	//******************** SCHEDA IN AP200.8
	I_AP200_8 			AT %I*: ARRAY[1..16] OF BOOL;
	//I_FREE 				: bool; // 1 = FREE
	//I_FREE 				: bool; // 2 = FREE
	//I_FREE 				: bool; // 3 = FREE
	//I_FREE 				: bool; // 4 = FREE
	I_24VOK_PS308			: BOOL;	// 5 = Presenza 24V PS308
	I_24VOK_PS309			: BOOL;	// 6 = Presenza 24V PS309
	I_24VOK_JB314			: BOOL;	// 7 = Presenza 24V JB314
	I_24VOK_JB315			: BOOL;	// 8 = Presenza 24V JB315
	//I_PresenzaSupporto[5] : BOOL;	// 9 = 
	//I_PresenzaTelaio[5]	: BOOL;	// 10 = 
	//I_PresenzaCentrale[5]	: BOOL;	// 11 = 
	//I_PresenzaBundle[5] 	: BOOL; // 12 = 
	//I_PresenzaSupporto[6] : BOOL;	// 13 = 
	//I_PresenzaTelaio[6]	: BOOL;	// 14 = 
	//I_PresenzaCentrale[6]	: BOOL;	// 15 = 
	//I_PresenzaBundle[6] 	: BOOL; // 16 =

	//******************** SCHEDA IN SAFETY AP200.9		
	I_AP200_9	AT %I*: ARRAY[1..4] OF BOOL;
	I_RicevitoreConsensoVeicolo AT %I*: ARRAY[1..8] OF BOOL;
	//I_RicevitoreConsensoVeicolo[1]	: BOOL; // 1=
	//I_RicevitoreConsensoVeicolo[2] 	: BOOL; // 2=	
	//I_RicevitoreConsensoVeicolo[3]	: BOOL; // 3=	
	//I_RicevitoreConsensoVeicolo[4]	: BOOL; // 4=	
	
	//******************** SCHEDA IN SAFETY AP200.10		
	I_AP200_10	AT %I*: ARRAY[1..4] OF BOOL;
	I_RichiestaIngressoPS308 			AT %I* : BOOL; // 2 = Richiesta ingresso Pal PS308
	I_ResetRichiestaIngressoPS308 		AT %I* : BOOL; // 6 = Richiesta ingresso Pal PS308
	//I_BarrieraCentroDx_CH1			: BOOL; // 3=	
	//I_BarrieraCentroDx_CH2			: BOOL; // 4=	

	//******************** SCHEDA IN SAFETY AP201.2		
	I_AP201_2	AT %I*: ARRAY[1..4] OF BOOL;
	//I_FeedBackMarcia				: BOOL; // 1=
	I_ResetRichiestaIngressoPS309 				AT %I* : BOOL; // 6 = Richiesta ingresso Pal PS309
	//I_BarrieraInterna_CH1			: BOOL; // 3=	
	//I_BarrieraInterna_CH2			: BOOL; // 4=	

	//******************** SCHEDA OUT AP201.4
	O_AP201_4 			AT %Q*: ARRAY[1..16] OF BOOL;		
	O_SirenaAllarmiPal							: BOOL;	// 1 = Sirena Allarmi
	O_LampadaAutomaticoPal						: BOOL;	// 2 = Lampada AUtomatico
	O_LampadaAllarmiPal							: BOOL;	// 3 = Lampada Allarmi
	O_LampadaRichiestaIngressoPal				: BOOL;	// 4 = Lampada Richiesta Ingresso PAL 1
	O_ConsensoVeicolo 							: ARRAY[1..8] OF BOOL;
	//O_ConsensoVeicolo[1]						: BOOL;	// 5 =
	//O_ConsensoVeicolo[2]						: BOOL;	// 6 =
	//O_ConsensoVeicolo[3]						: BOOL;	// 7 =
	//O_ConsensoVeicolo[4]						: BOOL;	// 8 =
	O_LampadaPulsanteCicloPalConsolle 			: BOOL;	//9 = Lampada Pulsante Ciclo Pallettizzatore
	O_LampadaPulsanteRichiestaIngressoConsolle 	: BOOL; //10 = Lampada Pulsante richiesta ingresso PS305
	O_LampadaPulsanteMarciaPalConsolle 			: BOOL;	//11 = Lampada Pulsante Marcia Pal 1 Consolle
	O_LampadaPulsanteRichiestaIngressoPS306 	: BOOL; //12 = Lampada Pulsante richiesta ingresso PS306
	O_LampadaPulsanteRichiestaIngressoPS307		: BOOL; //13 = Lampada Pulsante richiesta ingresso PS307
	O_LampadaPulsanteRichiestaIngressoPS308 	: BOOL; //14 = Lampada Pulsante richiesta ingresso PS308
	O_LampadaPulsanteRichiestaIngressoPS309		: BOOL; //15 = Lampada Pulsante richiesta ingresso PS309
	//FREE 										: BOOL; //16 =

	//******************** SCHEDA OUT SAFETY AP201.5		
	O_AP201_5	AT %Q*: ARRAY[1..4] OF BOOL;  			I_AP201_5 AT %I*: ARRAY[1..4] OF BOOL;//Appoggio
	//O_MarciaPal	: BOOL; // CH1=
	//FREE			: BOOL; // CH2=	
	//FREE			: BOOL; // CH3=	
	//FREE			: BOOL; // CH4=	
	
	//******************** SCHEDA OUT AP201.6	
	O_AP201_6 						AT %Q*: ARRAY[1..16] OF BOOL;
	
	O_LampadaIngressoVietatoPS306 	: BOOL; // 1 = Lampada Pulsante richiesta ingresso PS306
	O_LampadaIngressoVietatoPS307 	: BOOL; // 2 = Lampada Pulsante richiesta ingresso PS306
	O_LampadaIngressoVietatoPS308 	: BOOL; // 3 = Lampada Pulsante richiesta ingresso PS306
	O_LampadaIngressoVietatoPS309 	: BOOL; // 4 = Lampada Pulsante richiesta ingresso PS306
	//O_ConsensoVeicolo[5]		  	: BOOL;	// 5 =
	//O_ConsensoVeicolo[6]			: BOOL;	// 6 =
	//O_ConsensoVeicolo[7]			: BOOL;	// 7 =
	//O_ConsensoVeicolo[8]			: BOOL;	// 8 =
	//FREE 							: BOOL; // 9 =
	//FREE 							: BOOL; // 10 =
	//FREE 							: BOOL; // 11 =
	//FREE 							: BOOL; // 12 =
	//FREE 							: BOOL; // 13 =
	//FREE 							: BOOL; // 14 =
	//FREE 							: BOOL; // 15 =
	//FREE 							: BOOL; // 16 =

	//******************** SCHEDA IN AP201.3	
	I_AP201_3 			AT %I*: ARRAY[1..16] OF BOOL;
		
	//I_PresenzaSupporto[7] : BOOL;	// 1 = 
	//I_PresenzaTelaio[7]	: BOOL;	// 2 = 
	//I_PresenzaCentrale[7]	: BOOL;	// 3 = 
	//I_PresenzaBundle[7] 	: BOOL; // 4 = 
	//I_PresenzaSupporto[8] : BOOL;	// 5 = 
	//I_PresenzaTelaio[8]	: BOOL;	// 6 = 
	//I_PresenzaCentrale[8]	: BOOL;	// 7 = 
	//I_PresenzaBundle[8] 	: BOOL; // 8 = 
	//FREE 							: BOOL; // 9 =
	//FREE 							: BOOL; // 10 =
	//FREE 							: BOOL; // 11 =
	//FREE 							: BOOL; // 12 =
	//FREE 							: BOOL; // 13 =
	//FREE 							: BOOL; // 14 =
	//FREE 							: BOOL; // 15 =
	//FREE 							: BOOL; // 16 =

	//******************** SCHEDA IN SAFETY AP202.2		
	I_AP202_2	AT %I*: ARRAY[1..4] OF BOOL;
	//I_RicevitoreConsensoVeicolo[5]	: BOOL; // 1=
	//I_RicevitoreConsensoVeicolo[6] 	: BOOL; // 2=	
	//I_RicevitoreConsensoVeicolo[7]	: BOOL; // 3=	
	//I_RicevitoreConsensoVeicolo[8]	: BOOL; // 4=	

	//******************** SCHEDA IN SAFETY AP202.3		
	I_AP202_3	AT %I*: ARRAY[1..4] OF BOOL;
	I_PresenzaVeicolo : ARRAY[1..8] OF BOOL;
	//I_PresenzaVeicolo[1]	: BOOL; // 1=
	//I_PresenzaVeicolo[2] 	: BOOL; // 2=	
	//I_PresenzaVeicolo[3]	: BOOL; // 3=	
	//I_PresenzaVeicolo[4]	: BOOL; // 4=	

	//******************** SCHEDA IN SAFETY AP202.5		
	I_AP202_5	AT %I*: ARRAY[1..4] OF BOOL;
	//I_PresenzaVeicolo[5]	: BOOL; // 1=
	//I_PresenzaVeicolo[6] 	: BOOL; // 2=	
	//I_PresenzaVeicolo[7]	: BOOL; // 3=	
	//I_PresenzaVeicolo[8]	: BOOL; // 4=	

	//******************** SCHEDA IN SAFETY AP202.6		
	I_AP202_6	AT %I*: ARRAY[1..4] OF BOOL;
	//I_BarrieraCentroSx_CH1	: BOOL; // 1=
	//I_BarrieraCentroSx_CH2 	: BOOL; // 2=	
	//I_BarrieraSx_CH1			: BOOL; // 3=	
	//I_BarrieraSx_CH2			: BOOL; // 4=	
	
	I_PHPresenzaPallet		: ARRAY[1..MAXAREA] OF BOOL; // Presenza pallet
	
END_VAR

// ---- Global Variables/TFVariable/Supervisor_Variable.TcGVL
{attribute 'Tc2GvlVarNames'}
VAR_GLOBAL
	HMI_ReqCambioWorkOrder      : BOOL; (* Bit che si alza per indicare a HMI la richiesta di un cambio di W.O.*)
	HMI_ConfermaCambioWorkOrder : BOOL; (* Conferma da operatore su HMI per cambio Workorder *)
	LGV_Data 					: ARRAY[1..MAXAREA] OF ST_SupervisorData;		//Dati per supervisore
	
END_VAR
VAR_GLOBAL PERSISTENT
	
	Request_WorkOrder 	: ST_WorkOrder; 	(* Nuovo ordine di lavoro - SCRITTO DA WMS *)
	
	ReadyToChange		: BOOL; 			(* Indica che la macchina è pronta a eseguire il cambio di produzione - SCRITTO DA PLC *)
	Actual_WorkOrder	: ST_WorkOrder;		(* Ordine di lavoro in esecuzione - SCRITTO DA PLC *)
	
	OLD_Actual_WorkOrder : ST_WorkOrder;	(* Ultimo Ordine di lavoro in esecuzione prima del cambio *)

	HMI_CambioOrdineAutomatico 	: BOOL := TRUE; (* Se TRUE l'ordine viene attivato autoomaticamente *) 
	StatisticData				:  ST_StatisticData;
END_VAR

// ---- Global Variables/TFVariable/TFGlobal.TcGVL
{attribute 'Tc2GvlVarNames'}
VAR_GLOBAL CONSTANT
	Pos0TrasporteCavallete						: UINT := 0;		
	Pos180TrasporteCavallete					: UINT := 180;	
	RIBALTINO_NOP								: INT := 0;
	RIBALTINO_VERTICALE							: INT := 1;
	RIBALTINO_ORRIZZONTALE						: INT := 2;
	
	NO_INTERPOLAZIONE_ASSE 						: INT := 0; (* Indica che l'interpolazione dell'asse non è abilitata *)
	INTERPOLAZIONE_ASSE 						: INT := 1; (* Indica che l'interpolazione dell'asse è abilitata *)
	INTERPOLAZIONE_VIRTUALE_VIRTALE				: INT := 2; (* Indica che è abilitata l'interpolazione "Virtuale" dell'asse *)
	
	(* Tipo HOMING *)
	HOMING_STANDARD				: INT := 1;//Indica l'homing standard con l'uso del sensore
	HOMING_TORQUE				: INT := 2;//Indica l'homing con l'uso del limite di coppia e controllo dell'errore di inseguimento

	(* Tipi di Encoder *)
	HOMING_ASSE_PINZA    	: INT := 4; //indica il reset x l'asse K quando si fa il cambio manipolatori
		
	SupportoVuoto 			: TFMachinePalletizer_Pallet;
	
	
END_VAR

VAR_GLOBAL
	(* Project Machine *)
	MachinePalletizer_TF : TFMachinePalletizer_TF;
	
	(* Project Modules *)
	//ModuloAsse_X 		: TFModulePalletizer_Ax;
	//ModuloAsse_Y 		: TFModulePalletizer_Ax;
	//ModuloAsse_Z 		: TFModulePalletizer_Ax;
	//ModuloAsse_K 		: TFModulePalletizer_Ax;
	//ModuloAsse_J 		: TFModulePalletizer_Ax;
	//ModuloAspirazione	: TFModulePalletizer_Aspirazione;

	MachinePalletizerModules	: TFPalletizerModules; //Moduli della macchina
	
	Ciclo_Di_Riposo				: Stato_Ciclo_Lavoro;
	Ciclo_Pelievo_Falda			: Stato_Ciclo_Lavoro;
	Ciclo_Deposito_Falda		: Stato_Ciclo_Lavoro;
	//Ciclo_Pelievo_Pallet		: Stato_Ciclo_Lavoro;
	//Ciclo_Deposito_Pallet		: Stato_Ciclo_Lavoro;
	Ciclo_Prelievo_Lastra		: Stato_Ciclo_Lavoro;
	Ciclo_Deposito_Lastra		: Stato_Ciclo_Lavoro;
	
	//Depallettizzatore
	Ciclo_Prelievo_Lastra_Depal		: Stato_Ciclo_Lavoro;
	Ciclo_Deposito_Lastra_Depal		: Stato_Ciclo_Lavoro;
	Ciclo_Deposito_Falda_Depal		: Stato_Ciclo_Lavoro;

	
	PacchiPrelevatiAlMinuto		: UINT;
	PacchiAlMinuto 				: ARRAY[1..50] OF UINT;
	PacchiPrelevatiIn5Minuti 	: REAL;
	TempoUltimoDeposito		 	: UINT;
	
	QuotaAnticipoDinamicaX_Raggiunta : BOOL;	//Se TRUE indica che la quota dell'asse X permette i movimenti sucessivi dei vari assi
	QuotaAnticipoDinamicaY_Raggiunta : BOOL;	//Se TRUE indica che la quota dell'asse Y permette i movimenti sucessivi dei vari assi
	QuotaAnticipoDinamicaZ_Raggiunta : BOOL;	//Se TRUE indica che la quota dell'asse Z permette i movimenti sucessivi dei vari assi
	QuotaAnticipoDinamicaJ_Raggiunta : BOOL;	//Se TRUE indica che la quota dell'asse J permette i movimenti sucessivi dei vari assi
	//QuotaAnticipoDinamicaK_Raggiunta : BOOL;	//Se TRUE indica che la quota dell'asse K permette i movimenti sucessivi dei vari assi
	
	QuotaX_ConsensoRotazionePinza_Raggiunta : BOOL;		//Se TRUE indica che l'asse X è alla quota in cui è possibile roto-traslare i vari assi senza rischiare di collidere con le colonne
	//ConsensoTraslazioneY_TraColonne 		: BOOL;
	IngombroSuperficialePinzaMAX_Global 	: LREAL;	//Ingombro Superficiale Massimo della pinza 
	IngombroXPinzaOttimizzato_Global 		: LREAL;	//Ingombro Ottimizzato della pinza in direzione X
	IngombroYPinzaOttimizzato_Global 		: LREAL;	//Ingombro Ottimizzato della pinza in direzione Y
	
	AreaInLavoroPositiva 			: BOOL;	//Indica che la piazzola di deposito e prelivo sono nella stessa zona di lavoro (a DX o SX delle colonne)
	AreaInLavoroNegativa 			: BOOL;	//Indica che la piazzola di deposito e prelivo sono nella stessa zona di lavoro (a DX o SX delle colonne)
	AreaInLavoroPositivaNegativa 	: BOOL;	//Indica che la piazzola di deposito e prelivo NON sono nella stessa zona di lavoro (DEVO PASSARE IN MEZZO ALLE COLONNE)

	WorkAreaDX_Attuale : UINT;
	WorkAreaSX_Attuale : UINT;
	
	QuotaAnticipoDinamicaX_DepositoPacco 	: LREAL;
	QuotaAnticipoDinamicaX_DepositoPallet 	: LREAL;
	QuotaAnticipoDinamicaZ_VersoDepPallet 	: LREAL;
	
	QuotaAnticipoDinamicaZ_VersoPrelPacco 	: LREAL;
	QuotaAnticipoDinamicaX_VersoDepPacco 	: LREAL;
	
	QuotaAnticipoDinamicaZ_VersoPrelPall 	: LREAL;
	QuotaAnticipoDinamicaX_VersoDepPall 	: LREAL;
	
	QuotaAnticipoDinamicaZ_VersoPrelFalda 	: LREAL;
	QuotaAnticipoDinamicaX_VersoDepFalda 	: LREAL;
	
	QuotaAnticipoDinamicaZ_VersoRiposo 		: LREAL;
	
	RibaltinoExitOk : BOOL; //Consenso al prelievo dal ribaltino
	
	STARTInterpolazioneASSI : BOOL;
	
	ProgrammaToModule_X_Interpolato : Descrittore_Programma;
	ProgrammaToModule_Y_Interpolato : Descrittore_Programma;
	ProgrammaToModule_Z_Interpolato : Descrittore_Programma;
	ProgrammaToModule_J_Interpolato : Descrittore_Programma;
	//ProgrammaToModule_K_Interpolato : Descrittore_Programma;
	
	Asse_X_InFinestraDiPassMode : BOOL;
	Asse_Y_InFinestraDiPassMode : BOOL;
	Asse_Z_InFinestraDiPassMode : BOOL;
	Asse_J_InFinestraDiPassMode : BOOL;
	//Asse_K_InFinestraDiPassMode : BOOL;
	
	EncoderEsternoAsse_X : GestioneEncoderEsterno; //Istanza Encoder  Assoluto Asse X
	//EncoderEsternoAsse_Y : GestioneEncoderEsterno; //Istanza Encoder  Assoluto Asse Y
	//EncoderEsternoAsse_Z : GestioneEncoderEsterno; //Istanza Encoder  Assoluto Asse Z
	//EncoderEsternoAsse_J : GestioneEncoderEsterno; //Istanza Encoder  Assoluto Asse J	
	//EncoderEsternoAsse_K : GestioneEncoderEsterno; //Istanza Encoder  Assoluto Asse K
	
	ArrayPacchiSIMULATO : DUT_ArrayPacchi;
	
	PaccoPresoXDataLogger : BOOL; //Variabile per loggare il numero di prese
	
	ApprendimentoNullo : TFMachinePalletizer_CoordinateApprendimento;
	
	EnablePneumatica : BOOL;//Abilitazione marcia pneumatica
	
	LOCAL_AmsNetId : T_AmsNetID;
	
	ResetNecessarioCentralinaSafety : BOOL;

	FuoriIngombroXNecessario : BOOL;//Indica che la macchina prima di muoversi deve portarsi in  fuori ingombro con l'asse X
	FuoriIngombroYNecessario : BOOL;//Indica che la macchina prima di muoversi deve portarsi in  fuori ingombro con l'asse Y
	FuoriIngombroZNecessario : BOOL;//Indica che la macchina prima di muoversi deve portarsi in  fuori ingombro con l'asse Z
	FuoriIngombroJNecessario : BOOL;//Indica che la macchina prima di muoversi deve portarsi in  fuori ingombro con l'asse J

(* Quote Fuoringobro *)
	QuotaFuoriIngombro_Z_ConPEZZO 	: LREAL; 
	QuotaFuoriIngombro_Z_ConPALLET 	: LREAL;
	QuotaFuoriIngombro_Z_ConFALDA 	: LREAL;

	//	
	QuotaFuoriIngombro_X_AVUOTO  	: LREAL;
	QuotaFuoriIngombro_Y_AVUOTO  	: LREAL;
	QuotaFuoriIngombro_Z_AVUOTO  	: LREAL;
	QuotaFuoriIngombro_J_AVUOTO  	: LREAL;

	//
	QuotaFuoriIngombro_X_ConCARICO 	: LREAL; 
	QuotaFuoriIngombro_Y_ConCARICO 	: LREAL; 
	QuotaFuoriIngombro_Z_ConCARICO 	: LREAL; 
	QuotaFuoriIngombro_J_ConCARICO 	: LREAL; 
	
	//
	QuotaFuoriIngombro_Z_AVUOTO_CCENTRALE	: LREAL;
	QuotaFuoriIngombro_Z_AVUOTO_CESTERNO  	: LREAL;
	QuotaFuoriIngombro_Z_AVUOTO_CINTERNO  	: LREAL;

	
	Quota_Attesa_Caduta_Falda_Z     			: LREAL;
	QuotaFUPRINGOMBROdaRIBALTINO_X_RAGGIUNTA 	: BOOL; //Indica che la pinza è in fuori ingombro col ribaltino in direzione X
	QuotaFUPRINGOMBROdaRIBALTINO_Y_RAGGIUNTA 	: BOOL; //Indica che la pinza è in fuori ingombro col ribaltino in direzione Y
	QuotaFuoriIngombroColonne_Y					: LREAL; //Quota Y di Fuori ingombro colonne 
	
	Pinza_InIngombroColonne_Attuale				: BOOL;//Indica che la pinzza si trova ini ingombro colonne alla partenza del ciclo
	Pinza_InIngombroColonne_Destinazione		: BOOL;//Indica che la pinzza si trova ini ingombro colonne alla fine del ciclo
	
	AsseXInFinestraDiPrelievo : BOOL;
	AsseYInFinestraDiPrelievo : BOOL; 
	AsseZInFinestraDiPrelievo : BOOL; 
	AsseJInFinestraDiPrelievo : BOOL;
	
	AsseXInIngombroColonnePerRotazione : BOOL;
	AsseYInIngombroColonnePerRotazione : BOOL;

	//Ingombro della pinza nelle varie dimensioni
	IngombroX_Pos : LREAL;//Ingombro ATTUALE della pinza nella Metà POSITIVA della pinza lungo X
	IngombroY_Pos : LREAL;//Ingombro ATTUALE della pinza nella Metà POSITIVA della pinza lungo Y
	IngombroZ_Pos : LREAL;//Ingombro ATTUALE della pinza nella Metà POSITIVA della pinza lungo Z
	
	IngombroX_Neg : LREAL;//Ingombro ATTUALE della pinza nella Metà NEGATIVA della pinza lungo X
	IngombroY_Neg : LREAL;//Ingombro ATTUALE della pinza nella Metà NEGATIVA della pinza lungo Y
	IngombroZ_Neg : LREAL;//Ingombro ATTUALE della pinza nella Metà NEGATIVA della pinza lungo Z
	
	IngombroDestinazioneX_Pos : LREAL;//Ingombro della pinza nella Metà POSITIVA della pinza lungo X
	IngombroDestinazioneY_Pos : LREAL;//Ingombro della pinza nella Metà POSITIVA della pinza lungo Y
	
	IngombroDestinazioneX_Neg : LREAL;//Ingombro della pinza nella Metà NEGATIVA della pinza lungo X
	IngombroDestinazioneY_Neg : LREAL;//Ingombro della pinza nella Metà NEGATIVA della pinza lungo Y
	
	IngombroDestinazioneZ_Pos : LREAL;//Ingombro della pinza lungo Z Positivo (sopra al fulcro)
	IngombroDestinazioneZ_Neg : LREAL;//Ingombro della pinza lungo Z Negativo (sotto al fulcro)
	
	IngombroMaxX_Pos : LREAL;//Ingombro MASSIMO della pinza nella Metà POSITIVA della pinza lungo X
	IngombroMaxY_Pos : LREAL;//Ingombro MASSIMO della pinza nella Metà POSITIVA della pinza lungo Y
	
	IngombroMaxX_Neg : LREAL;//Ingombro MASSIMO della pinza nella Metà NEGATIVA della pinza lungo X
	IngombroMaxY_Neg : LREAL;//Ingombro MASSIMO della pinza nella Metà NEGATIVA della pinza lungo Y
	
	IngombroMaxZ_Pos : LREAL;//Ingombro MASSIMO della pinza lungo Z Positivo (sopra al fulcro)
	IngombroMaxZ_Neg : LREAL;//Ingombro MASSIMO della pinza lungo Z Negativo (sotto al fulcro)

	IngombroY_Pos_0 	: POINTER TO LREAL;//Ingombro della pinza nella Metà POSITIVA della pinza lungo Y nella posizione 0°
	IngombroY_Neg_180 	: POINTER TO LREAL;//Ingombro della pinza nella Metà NEGATIVA della pinza lungo Y nella posizione 180°
	IngombroY_Neg_0 	: POINTER TO LREAL;//Ingombro della pinza nella Metà POSITIVA della pinza lungo Y nella posizione 0°
	IngombroY_Pos_180 	: POINTER TO LREAL;//Ingombro della pinza nella Metà NEGATIVA della pinza lungo Y nella posizione 180°

	ScostamentoVerticalePuntoCentrale : LREAL; //Valore dhe rappresenta quanto il punto centrale si è spostato rispetto allo zero orizzontale (lungo Z crescente)	

	IngombroZ : LREAL;//Ingombro della pinza lungo Z
	
	IngombroY_Tot : LREAL;//Ingombro in direzione Y

	SupportoSvuotatoLato90 		: ARRAY[1..MAXAREA] OF BOOL; //Array indicante supporti terminati
	SupportoSvuotatoLato0 		: ARRAY[1..MAXAREA] OF BOOL; //Array indicante supporti terminati
	SupportoSvuotatoLato180 	: ARRAY[1..MAXAREA] OF BOOL; //Array indicante supporti terminati

	MaterialeDepositatoSuLinea 	: BOOL;//Segnalazione di materiale depositato a MP
	SchedulerIDSuPinza 			: DWORD;	
	
	MemoriaQuoteTasteggio 		: ARRAY[1..10] OF REAL;//arrey memoria di quote tasteggio, serve per determinare se evacuare o meno il pallet
	MemoriaQuoteTasteggioVuoto	: ARRAY[1..10] OF REAL;
	idxTasteg 					: UINT;//Indice usato per riempire l'array di memoria delle quote di tasteggio
	StopDepositoPerArresto 		: BOOL; //Memoria di richiesta stop ciclo deposito su rulliera
	TFCalcoloFormatura 			: Calcolo_Formatura_Completa;//FB per il calcolo della formatura
	TFCalcoloFormaturaDaLista	: Calcolo_Formatura_Completa;//FB per il calcolo della formatura
	TFCalcoloFormaturaRT		: ARRAY[1..3] OF Calcolo_Formatura_Completa;//FB per il calcolo della formatura
	TFCalcoloFormaturaEmpty		: Calcolo_Formatura_Completa;//FB per il calcolo della formatura

	SIMULAZIONE_NO_HW 				: BOOL:= FALSE;
	FormingEmpty 				: TFMachinePalletizer_FormingForSlab;
	FaldaDaDepositare : TFMachinePalletizer_PlaceElement;//Descrizione falda da depositare, valorizzata dal WorkOrder
	
	SupportDataEmpty : ST_SupportData;

//#### Variabili per Test
	M255 						: BOOL := TRUE; 			//# RIcorda Forzatura
	M255_sempreON 				: BOOL := TRUE;
	M255_sempreOFF 				: BOOL := FALSE;
	
	
//##
	CoordenadaZInicial: REAL;

	In_PosRobot								: UINT;
	PosRobot								: UINT;
	QuotaCentroPostazioneIni				: LREAL;
	QuotaCentroPostazionePiking				: LREAL;
	PosicionJActual							: LREAL;
	RobotWorkAreaCavallete 					: BOOL ;
	RobotCentroPosX							: BOOL ;
	CotaCentroPosRobot						:LREAL ;
	
	PosicionJDestino						: LREAL;
	PosicionJOrigen							: LREAL;
	EjeYPosFueraIngombro					: BOOL;
	EjeYPos0Ingombro						: BOOL;
	EjeYPos180Ingombro						: BOOL;
	EjeyPosLentaCoger						: BOOL ;
	Z_PuntoPrelievo180Bundle				: LREAL;
	
//##Depuracion Alberto
	NuIngombroYCalculado180G_Depuracion		: UINT ;
	NuIngombroYCalculado0G_Depuracion		: UINT ;
	NuIngombroYCalculado90G_Depuracion		: UINT ;
	
	Ok_sensores_Tastator: BOOL;
	Nu_Sensores_Leyendo: BYTE;
	// Habilitacion Giro coger con fc
	Habilito_Pos_j_Fc: BOOL;
	EjexEnPosicion: LREAL;
END_VAR

VAR_GLOBAL PERSISTENT

	(* Parametri nominali degli assi - Coincidenti con i parametri presenti nella scheda NC *)
	AxisNominalPar_X			: Ax_Palletizer_Nominal_Parameters;
	AxisNominalPar_Y			: Ax_Palletizer_Nominal_Parameters;
	AxisNominalPar_Z			: Ax_Palletizer_Nominal_Parameters;
	AxisNominalPar_J			: Ax_Palletizer_Nominal_Parameters;
	//AxisNominalPar_K			: Ax_Palletizer_Nominal_Parameters;
	
	(* Parametri degli assi *)
	AxisPar_X					: Ax_Palletizer_Parameters;
	AxisPar_Y					: Ax_Palletizer_Parameters;
	AxisPar_Z					: Ax_Palletizer_Parameters;
	//AxisPar_K					: Ax_Palletizer_Parameters;
	AxisPar_J					: Ax_Palletizer_Parameters;
	
	AxisHomingParameters_X		: AxHomingParameters;	
	AxisHomingParameters_Y		: AxHomingParameters;	
	AxisHomingParameters_Z		: AxHomingParameters;	
	AxisHomingParameters_J		: AxHomingParameters;	
	//AxisHomingParameters_K		: AxHomingParameters;	
	(* Override degli assi *)
	AxisOverride				: TFMachinePalletizer_VelocityOverride_TF;
	
	ProgrammaToModule_X			: Descrittore_Programma;
	ProgrammaToModule_Y			: Descrittore_Programma;
	ProgrammaToModule_Z			: Descrittore_Programma;
	ProgrammaToModule_K			: Descrittore_Programma;
	ProgrammaToModule_J			: Descrittore_Programma;
	
	ProgrammaToModuleNEXT_X		: Descrittore_Programma;
	ProgrammaToModuleNEXT_Y		: Descrittore_Programma;
	ProgrammaToModuleNEXT_Z		: Descrittore_Programma;
	ProgrammaToModuleNEXT_K		: Descrittore_Programma;
	ProgrammaToModuleNEXT_J		: Descrittore_Programma;

	(* Stato dei moduli *)
	Status_TF 							: TFModulePalletizerSTATUS_TF;
	(* Parametri assi : Velocità/ Accelerazioni / Decelerazioni CON e SENZA carico relativi ai vari programmi *)
	ParametriProgramma_X_CicloRiposo	: Ax_Program_Parameters;
	ParametriProgramma_Y_CicloRiposo	: Ax_Program_Parameters;
	ParametriProgramma_Z_CicloRiposo	: Ax_Program_Parameters;
	ParametriProgramma_J_CicloRiposo	: Ax_Program_Parameters;
	//ParametriProgramma_K_CicloRiposo	: Ax_Program_Parameters;
	
	ParametriProgramma_X_CicloPallet	: Ax_Program_Parameters;
	ParametriProgramma_Y_CicloPallet	: Ax_Program_Parameters;
	ParametriProgramma_Z_CicloPallet	: Ax_Program_Parameters;
	ParametriProgramma_J_CicloPallet	: Ax_Program_Parameters;
	//ParametriProgramma_K_CicloPallet	: Ax_Program_Parameters;
	
	ParametriProgramma_X_CicloFalda		: Ax_Program_Parameters;
	ParametriProgramma_Y_CicloFalda		: Ax_Program_Parameters;
	ParametriProgramma_Z_CicloFalda		: Ax_Program_Parameters;
	ParametriProgramma_J_CicloFalda		: Ax_Program_Parameters;
	//ParametriProgramma_K_CicloFalda		: Ax_Program_Parameters;

	ParametriProgramma_X_CicloLastra		: Ax_Program_Parameters;
	ParametriProgramma_Y_CicloLastra		: Ax_Program_Parameters;
	ParametriProgramma_Z_CicloLastra		: Ax_Program_Parameters;
	ParametriProgramma_J_CicloLastra		: Ax_Program_Parameters;
	//ParametriProgramma_K_CicloLastra		: Ax_Program_Parameters;
	(* Traiettoria *)
	Traiettoria 						: TFTraiettoria;
	(* Gestore degli stati delle WORKAREA *)
	WorkAreaManager						: TFWorkAreaManager;
	(* Stati delle missioni *)
	MissionStateCase					: MissionStateCase;
		
	(* Variabili per punto di riposo *)
	X_Riposo	: LREAL;
	Y_Riposo	: LREAL;
	Z_Riposo	: LREAL;
	J_Riposo	: LREAL;
	K_Riposo	: LREAL;
	
	Dimensione_Z_ElementoInPresaX_Ingombro : REAL; // E' la somma della dimensione che ha l'ogetto in presa sulla pinza (Pallet/Falda/Pacco) + eventuali offest di prelievo.. in modo da avere l'ingombro Verticale REALE!! dell'oggetto..
	
	Dimensioni_Pinza	:	TFDimensioniPinza;
	
	(* Offset sicurezza movimenti *)
	OffsetSicurezzaAnticipoMovimenti	: Offset_Sicurezza_Anticipo_Movimenti;
	OffsetSicurezza					 	: OffsetSicurezzaIngombro;
	OffsetPrelieviLenti				 	: Offset_Prelievi_Lenti;
	OffsetPassMode						: Offset_Pass_Mode;
	OffsetCadutaFalda				 	: REAL := 200;
	OffsetDistacco				 		: OffsetDistacco;
	
	(* Dimensioni Pick-Point *)
	WorkPickPointDimension : ARRAY[1..MAXPICKPOINT] OF Work_PickPoint_Dimension;
	
	PaccoSulRibaltino : TFHandlingPack;
	
	I_PHPresenzaPalletVirtuale :  ARRAY[1..MAXAREA] OF BOOL; //Simula la fotocellula di presenza pallet, utilizzato per i test senza HW
	
	InvertiComandoJog_X : BOOL := TRUE;
	InvertiComandoJog_Y : BOOL := FALSE;
	
	OffsetApprendimento : Offeset_Apprendimento;
	
	IDFormatura : UINT;
	GUIDFormatura : UINT;

	WorkAreaCodiciFissi : ARRAY [1..MAXAREA] OF INT;
	
	AmsNetId AT %I* : T_AmsNetIdArr;	
	OffSetPosYReposo 		:REAL := 230;
	//RetardoAlarTastatore :TON ; 
	
	
	
	
	Temp_Bool 	:ARRAY[0..100] OF BOOL;
	Temp_INT	:ARRAY[0..9] OF INT;
	Temp_UINT	:ARRAY[0..9] OF UINT;
	Temp_DINT	:ARRAY[0..9] OF DINT;
	Temp_UDINT	:ARRAY[0..9] OF UDINT;
	Temp_REAL	:ARRAY[0..9] OF REAL;
	Temp_LREAL	:ARRAY[0..9] OF LREAL;
	Temp_WORD	:ARRAY[0..9] OF WORD;			
	Temp_DWORD	:ARRAY[0..9] OF DWORD;
	Temp_SupportData : ARRAY[0..3] OF ST_SupportData; (* Dati del supporto in piano per legni*)	
	Temp_IdxLista : INT;
	Temp_i	: INT;
	LoopLista : UINT;
	ProgramaEjes 					: ProgramaEjecucion ;
	
	
	
	
	
	RetardoFcTastastatore 								: ARRAY [1..4] OF REAL ;
	RetardoFcTastastatoreJ								: ARRAY [1..2] OF REAL ;
	Re_TastatoreEmergenzaPinza							: ARRAY [1..4] OF REAL ;
	Re_In_TastatoreEmergenzaPinza						: ARRAY [1..4] OF BOOL ;
	Re_In_TastatorePinza								: ARRAY [1..4] OF BOOL ;
	RetardoTastatore 									:BOOL ;
	RetardoTastatoreJ 									:BOOL ;
	RegistroAlarma2205									:UINT ;
	RegistroCotaApolloY									:UINT ;
	TFFormacionBandelCalculada							: Calcolo_Formatura_Completa;//FB per il calcolo della formatura
	TFFormacionCavalleteCalculada						: Calcolo_Formatura_Completa;//FB per il calcolo della formatura
	TFCalcoloFormaturaWA								: ARRAY[1..MAXAREA] OF Calcolo_Formatura_Completa;//FB per il calcolo della formatura
	TipoLLenarCavellete									 :UINT := 4 ;
	ReControlPiezaCogida								: REAL ;
	
	OffSetZRecogidaEnAngulo0							: REAL ;
	OffSetZRecogidaEnAngulo180							: REAL ;
	
	PikingConCavallete									: BOOL ;
	AngulosDiferentes									: BOOL ;
	ReMovEjeX											: REAL ;
	ReMovEjeXCicloDeposito								: REAL ;
	AreaPikingConCavallete								: BOOL ;
	MultiplesCavalletesReceta							: BOOL ;
	NuEstacionesPiking									: UINT ;
	NuEstacionPiking									: UINT ;
	PosCavalleteOrdenPikin								: ARRAY [1..MAXAREA] OF e_Tipo_Pallet ;
	CoordenadaPasillo0_Y								: LREAL ;
	CoordenadaPasillo180_Y								: LREAL ;
	CoordenadaPosGiroPieza_X							: LREAL ;
	NuPosGuiroPiking									: UINT ;
	PIezaAgarrada										: BOOL ;
	WaCavalleteEnPiking									: INT;
	PosFinOrdenPikingCaballete							: UINT ;
	EjeYPosFueraIngombroCargado                         : BOOL;
	CuotaOffSetZRecogidaBundel							: LREAL ;
	CuotaOffSetZRecogidaCaballete						: LREAL ;
	GestionDescargaCaballete							: Es_LadosCaballete;
	GestionCargaCaballete								: Es_LadosCaballete;
	
	HabilitacionFormacionNueva							: BOOL;
	
	FormacionesCalculadas								: BOOL;
	FormacionPikingCalculada							: BOOL ;
	HabilitapikingPruevas								: BOOL;
END_VAR

// ---- Global Variables/TFVariable/TFMotion_Program.TcGVL
{attribute 'Tc2GvlVarNames'}
VAR_GLOBAL CONSTANT
	(* Numero di punti per il calcolo della traiettoria *)
	MAXTPOINTS : INT := 5; 
	(*STATI DEI PROGRAMMI*)
	NON_ESEGUITO 	: UINT := 0;
	DA_ESEGUIRE		: UINT := 1;
	IN_ESECUZIONE 	: UINT := 2;
	TERMINATO		: UINT := 3;
	INTERROTTO		: UINT := 4;
	ANNULLATO		: UINT := 5;
	TRASFERITO		: UINT := 6;
	(*Tipo Di Deposito*)
	DEPOSITO_FALDA_SU_CATASTA 	: UINT := 1;
	DEPOSITO_FALDA_SU_PIAZZOLA	: UINT := 2;
END_VAR

VAR_GLOBAL
	Programma_X : ARRAY[0..200] OF Descrittore_Programma;
	Programma_Y : ARRAY[0..200] OF Descrittore_Programma;
	Programma_Z : ARRAY[0..200] OF Descrittore_Programma;
	Programma_K : ARRAY[0..200] OF Descrittore_Programma;
	Programma_J : ARRAY[0..200] OF Descrittore_Programma;
END_VAR

// ---- Global Variables/TFMachinesErrors.TcGVL
{attribute 'Tc2GvlVarNames'}
VAR_GLOBAL CONSTANT

	(******************************************************************************************************************************************)
	(* Machine Errors *)
	(******************************************************************************************************************************************)
	ErrMACHINE_CPUSAFETYNOTOK 					: UINT := 2100; (* Machine - CPU Safety NOT Ok *)
	ErrMACHINE_CPUSAFETYNOTRUNNING 				: UINT := 2101; (* Machine - CPU Safety NOT Running *)
	ErrMACHINE_IOSAFETYNOTOK 					: UINT := 2102; (* Machine - IO Safety NOT Ok *)

END_VAR

// ---- Global Variables/TFMachinePalletizerVariables.TcGVL
{attribute 'Tc2GvlVarNames'}
VAR_GLOBAL CONSTANT

	MAXWORKFLOW : UINT := 12;//Numero di Workflow presenti

	(******************************************************************************************************************************************)
	(* Palletizer Constant *)
	(******************************************************************************************************************************************)
	MAXFOOTPRINT 								: UINT := 16; //Ingombri
	
	MAXPICKPOINT 								: UINT := 1; //Punti di prelievo
	
	MAXAREA 									: UINT := 12;//Piazzole di lavoro
	
	MAXPALLET 									: UINT := 32; //Numero di pallet
	
	MAXLAYER 									: UINT := 32; //Numero di falde
	
	MAXFORMINGCODE 								: UINT := 32; //Numero di codici di formatura
	
	MAXFORMINGPACK 								: UINT := 128; //Numero di pacchi in formatura
	
	MAXFORMING 									: UINT := 12; //Numero di formature attive contemporaneamente = NUMERO DI POSTAZIONI IN MACCHINA
	
	MAXZONE 									: UINT := 8; //Numero massimo numero di zone
	
	MAXHANDLINGPACK								: UINT := 15;
	
	MAXHANDLINGSTACK							: UINT := 8;
		
	MAXFORMINGSLAB	 							: UINT := 128;//Numero di Lastre/Elementi in Formatura
	
	PICKPOINT1									: UINT := 1;
	PICKPOINT2									: UINT := 2;
	PICKPOINT3									: UINT := 3;
	PICKPOINT4									: UINT := 4;
	
	KPRODUCTLOADING								: INT := 0;
	KPRODUCTLOADED								: INT := 1;
	KPRODUCTUNLOADING							: INT := 2;
	KPRODUCTUNLOADED							: INT := 3;
	KNOPRODUCT									: INT := 5;
	
	
	ZRESTPOSITION								: REAL := 1600.0;
	PICKLTRESTPOSITION							: INT  := 0; // LONGITUDINALE
 	VORESTPOSITION								: INT  := 0;
	KRESTPOSITION								: REAL := 700.0;
	TORQUERESTPOSITION							: REAL := 15;
	KPICKMODERESTPOSITION						: INT  := 1;
	
		
	OFFSETKPOSITION								: REAL := 40.0; //Quota fittizzia aggiuntiva per raggiungere la coppia necessaria in chiusura pinza
	OFFSETTORQUEPOSITION						: REAL := 40.0;
	KPICKTORQUELAYER							: REAL := 100.0;//Coppia per apertura/Chiusura Pinza in prelievo falda
		
	MAXSOGLIEOVERRIDE 							: UINT := 4;	// Numero di soglie utilizzate per il calcolo dell'override dinamico
	
	MAXNUMVISIONSYSTEM 		: INT := 3; //Indica il numero di sistemi di visione di difetti presenti

	MAXTYPE_SLABLAYER 		: UINT := 2; // Numero massimo di tipi di materiale (lastre o falde)

END_VAR
	
VAR_GLOBAL

	MachinePalletizerInitDone : BOOL := FALSE;
	MachinePalletizerInitVariables	: BOOL; (* Init Variables To Desired Values *)
	ParametersArray : ParametersArray;
	(* Variabile per Visualizzazione in debug *)
	l : INT;
	z : INT;
	
	(* Gate Access *)
	MachinePalletizerGatesAccess : TFMachinePalletizer_GatesAccess;
	(* Errori GATEACCESS *)
	GateAccessError							: UINT;
	(* Errori LGV *)
	LGVError 								: UINT;
	
	(* Project Modules I/O/Motion/Inverter *)	
	X_Axis									: AXIS_REF;
	X_AxisLib								: TFMotion;

	Y_Axis									: AXIS_REF;
	Y_AxisLib								: TFMotion;

	Z_Axis									: AXIS_REF;
	Z_AxisLib								: TFMotion;
	
	(* Rotazione Basculante Pinza - Angolo di Pitch *)
	J_Axis									: AXIS_REF;
	J_AxisLib								: TFMotion;
	(* Rotazione Piano Ventose Pinza - Angolo di Roll *)
	K_Axis									: AXIS_REF;
	K_AxisLib								: TFMotion;
	(* Rotazione Intero Corpo Pinza - Angolo di Yaw *)
	W_Axis									: AXIS_REF;
	W_AxisLib								: TFMotion;

	(* Change Gripper Configuration *)
	ChangeGripperConfig						: BOOL;
	
	(* Pallet and Layer stacks state *)
	PalletStackEmpty 						: INT;
	LayerStackEmpty 						: INT;
	AllWABusy								: INT;
	//EmptyPack                               : TFHandlingPack;
	EmptySlab                               : TFMachinePalletizer_PlaceElement;
	
	OSchedulerIDPerLinea AT %Q* 			: DWORD;//Scheduler ID doppia lunghezza per linea

	StatoMissione : INT := 0;//Stato della missione del pallettizzatore per segnalazione a HMI: 0=Nessuna Missione Attiva;1=Missione Attiva 
		
	FirstStatrtEx : BOOL;	

	NCodiciPresenti : UINT;// numero di codici presenti in fase di attivazione formatura
	
	EmptyWorkAreaState 	: TFMachinePalletizer_WorkAreaState;
	EmptySlabArray 		: ARRAY[1..MAXFORMINGSLAB] OF TFMachinePalletizer_PlaceElement;
	EmptyDataSlab       : ST_SlabData;
	EmptyDataSlabArray 	: ARRAY[1..MAXFORMINGSLAB] OF ST_SlabData;

	EseguitoAllinementoPezziDeposito : BOOL;//bit per impedire mescolamenti in fase di "annullamento" missione con stacco aspirazione
	
	NumeroPezziPresentiPostazioneStart : ARRAY[1..MAXAREA] OF UINT;//numero pezzi allo start della lavorazione
	
END_VAR

{attribute 'Tc2GvlVarNames'}
VAR_GLOBAL PERSISTENT
	
	WorkSpace 				: TFMachinePalletizer_WorkSpace;										(* Work Space (Spazio di Lavoro) *)
	WorkFootprint 			: ARRAY [1..MAXFOOTPRINT] OF TFMachinePalletizer_WorkFootprint;			(* Work Footprint (Ingombri "Parallelepipedi") *)
	WorkPickPoint 			: ARRAY [1..MAXPICKPOINT] OF TFMachinePalletizer_WorkPickPointSlab;			(* Work PickPoint (Punti di Prelievo Pacchi) *)
//WorkPickPointState 		: ARRAY [1..MAXPICKPOINT] OF TFMachinePalletizer_WorkPickPointState;	(* Work PickPoint State (Stato Punti di Prelievo Pacchi) *)
	WorkPickPointState		: ARRAY [1..MAXPICKPOINT] OF TFMachinePalletizer_WorkPickPoint_State;	(* Work PICKPOINT Roller State (Stato Punti di Prelievo Lastre: RULLIERE) *)
	//WorkPickPointTransportState : ARRAY [1..MAXPICKPOINT] OF TFMachinePalletizer_WorkPickPointTransport_State; (* Work PICKPOINT TRANSPORT State (Stato Punti di Prelievo Lastre traporti -> es. rulliere a terra ) *)


	//WorkPickPointStoreState	: POINTER TO ARRAY [1..MAXPICKPOINTSTORE] OF TFMachinePalletizer_WorkPickPointStore_State;	(* Work STORE State (Stato Punti di Prelievo STATICI: Magazzini: Layer,ecc) *)
	WorkPickPointOffset 	: ARRAY [1..MAXPICKPOINT] OF TFMachinePalletizer_WorkPickPointOffset;			(* Offset dei PickPoint rispetto le posizioni assolute *)
	
	
	
	
	WorkArea 				: ARRAY [1..MAXAREA] OF TFMachinePalletizer_WorkArea;					(* Work Area (Postazioni Pallet/Vuoti/Falde) *)
	WorkAreaState 			: ARRAY [1..MAXAREA] OF TFMachinePalletizer_WorkAreaState;				(* Work Area State (Stato Postazioni) *)
	WorkAreaOffset 			: ARRAY [1..MAXAREA] OF TFMachinePalletizer_WorkAreaOffset;				(* Offset delle postazioni rispetto le posizioni assolute *)
	WorkAreaZone			: TFMachinePalletizer_WorkAreaZone;										(* Suddivisione in zone delle postazioni del pallettizzatore  per gestire la priorità di deposito *)
	Pallet 					: ARRAY [1..MAXPALLET] OF TFMachinePalletizer_Pallet;					(* Pallet (Caratteristiche Pallet) *)
	Layer 					: ARRAY [1..MAXLAYER] OF TFMachinePalletizer_Layer;						(* Layer (Caratteristiche Falde) *)
	Forming 				: ARRAY [1..MAXFORMING] OF TFMachinePalletizer_FormingForSlab;					(* Layer (Caratteristiche Formatura) *)
	AxisPar					: TFModulePalletizerRobot_AxisPar;										(* Axis Parameters *)
	ManCmd					: TFModulePalletizerRobot_ManCmd;										(* Manual Commands *)
	Mission					: TFMachinePalletizer_Mission;											(* Missione della macchina *)
	MachineManCmd			: TFMachinePalletizer_ManCmd;											(* Comandi Manuali della Macchina *)
	PickPlaceParameters		: TFMachinePalletizer_PickPlaceParameters;								(* Parametri di prelievo e deposito *)
	TCPParameter			: TFModulePalletizerRobot_TCPPar;										(* Parametri del TCP (pinza) *)
	ProgressiveNrWA			: UDINT;																(* UDC delle postazioni:Aggiornato ad ogni deposito "Pallet"*)
	ProductOnGripper		: INT := KPRODUCTUNLOADED;												(* Indica cosa è presente nella pinza *)
	UsedCode				: ARRAY [1..MAXFORMINGCODE] OF INT;										(* Codici utilizzati *)
	GripperConfiguration	: INT;																	(* Indica il numero della configurazione della pinza *)
	(**********************************************************************************************************************************************************************************)
	(**********************************************************************************************************************************************************************************)
	PreviousPWA 			: INT;
	PreviousStackWA			: INT;
	RestoreCWA				: BOOL;
	TouchErrorEnable		: BOOL;																	(* Var Appoggio per Abilitazione Errore Tastatori *)
	(**********************************************************************************************************************************************************************************)
	(**********************************************************************************************************************************************************************************)
	IPalletizer_Safety_Gate_Enable : BOOL;
	(**********************************************************************************************************************************************************************************)
	(**********************************************************************************************************************************************************************************)
	Status					: TFModulePalletizerRobot_Status;	(* Indica lo stato del pallettizzatore *)
	(**********************************************************************************************************************************************************************************)
	(**********************************************************************************************************************************************************************************)
	AbilitazionePassModeGlobale : BOOL := TRUE; (* Abilitazione globale PassMode *)

	UltimaPostazioneInPrelievo : UINT;//Indica l'ultima postazione che è stata lavorata
	UltimoSchedulerLavorato : STRING;//Indica l'ultimo scheduler lavorato dalla macchina
	RichiestaCambioScheduler : BOOL;//Indica la richiesta all'operatore del cambio scheduler e attende la pressione del pulsante ciclo per partire
	UltimaTipologiaLavorata : INT;

	WorkAreaProductionList : ARRAY [1..MAXAREA] OF TFMachinePalletizer_ListaProduzione_WAM;
	WorkAreaStateBK	: ARRAY [1..MAXAREA] OF TFMachinePalletizer_WorkAreaState;
END_VAR

// ---- Global Variables/TFMachinePalletizerErrors.TcGVL
{attribute 'Tc2GvlVarNames'}
VAR_GLOBAL CONSTANT

	(******************************************************************************************************************************************)
	(* Machine Errors *)
	(******************************************************************************************************************************************)
	(* Machine Palletizer *)
	ErrMACHINEPALLETIZER_HOME_HSKTO							: UINT := 2103; (* Machine - Handshake Timeout From Preparing/Sewing Machine *)
	ErrMACHINEPALLETIZER_EMERGENCY							: UINT := 2104; (* Machine - Emergency not Ok *)
	ErrMACHINEPALLETIZER_PHASE380							: UINT := 2105; (* Machine - Phase 380 not Ok *)
	ErrMACHINEPALLETIZER_MAIN24V							: UINT := 2106; (* Machine - Main 24V not Ok *)
	ErrMACHINEPALLETIZER_MOTOR24V							: UINT := 2107; (* Machine - Motor 24V not Ok *)
	ErrMACHINEPALLETIZER_OUTPUT24V							: UINT := 2108; (* Machine - Output 24V not Ok *)
	ErrMACHINEPALLETIZER_DRIVE								: UINT := 2110; (* Machine - Drive not Ok *)
	ErrMACHINEPALLETIZER_CARTER								: UINT := 2111; (* Machine - Carter not Ok *)
	ErrMACHINEPALLETIZER_THERMAL							: UINT := 2112; (* Machine - Thermal not Ok *)
	ErrMACHINEPALLETIZER_CONDITIONER						: UINT := 2113; (* Machine - Conditioner not Ok *)
	ErrMACHINEPALLETIZER_AIR								: UINT := 2114; (* Machine - Air not Ok *)
	
	ErrMACHINEPALLETIZER_MISSINGPOWER						: UINT := 2116; (* Mancanza Marcia o almeno un asse senza Marcia *)
	
	ErrMACHINEPALLETIZER_BARRIEREOCCUPATE_LGVREQ_OFF			: UINT := 2117; (* Barriere di sicurezza occupate su riattivazione GateAccess dopo Ingresso TGV*)
	ErrMACHINEPALLETIZER_ANOMALIA_CONSENSI_SUPNAVETTE			: UINT := 2118; (* Avviene se ho un'anomalia della richiesta di ingresso e ingrombro dato dalla sup.Nav., solitamente in caso di manuale/emergenza della macchina *)
	ErrMACHINEPALLETIZER_AZZERAMENTO_FORZATO_RICHIN_SUPNAVETTE	: UINT := 2119; (* Avviene se ho UN ERRORE della macchina durante una richiesta di ingresso del TGV *)
    ErrMACHINEPALLETIZER_ERRORE_MACCHINA_IN_RICHIN				: UINT := 2120; (* Avviene se ho UN ERRORE della macchina durante una richiesta di ingresso *)
	
	ErrMACHINEPALLETIZER_PERDITARICHIAMATAPOST				: UINT := 2121;	(* Avviene se durante una richiesta di ingresso navetta si perde la CHIAMATA della postazione*)
	ErrMACHINEPALLETIZER_PERDITARICINGRESSOPOST				: UINT := 2122;	(* Avviene se durante una richiesta di ingresso navetta si perde la RICHIESTA DI INGRESSO nella postazione*)
	
	ErrMACHINEPALLETIZER_PHOFFDOPODEPOSITO					: UINT := 2122; (* Avviene dopo un DEPOSITO da parte della navetta, se la fotocellula non risulta essere accesa *)
	ErrMACHINEPALLETIZER_PHONDOPOPRELIEVO					: UINT := 2123; (* Avviene dopo un PRELIEVO da parte della navetta, se la fotocellula risulta essere accesa *)
	ErrMACHINEPALLETIZER_MANCATOAGGIORNAMENTOSTATO			: UINT := 2124; (* Avviene dopo un PRELIEVO/DEPOSITO da parte della navetta, se NON ha modificato lo stato della piazzola in Prelievo/Deposito effettuato*)
	

	ErrCONFIGURAZIONEPINZASABGLIATA				: UINT := 2189; (* Codice pallet o layer non trovato *)
	ErrMACHINEPALLETIZERTCALC					: UINT := 2190;	(* Machine - Trajectory Calculation Error *)
	ErrMACHINEPALLETIZERPACKPOINTERNOTVALID		: UINT := 2191; (* Machine - Pack Pointer Added is not valid *)
	ErrCYCLEPALLET								: UINT := 2192; (* Pallet Già Presente *)
	ErrCYCLELAYER								: UINT := 2193; (* Pallet non Presente *)
	ErrPACKCODEORDIMENSIONNOTVALID				: UINT := 2194; (* Codice o dimensioni Pacco presente su Ribaltino non Valide *)
	ErrPALLETORLAYERCODENOTFOUND				: UINT := 2195; (* Codice pallet o layer non trovato *)
	
	ErrPACKCODENOTVALID							: UINT := 2196; (* Codice Pacco presente su Ribaltino non Valide *)
	ErrPACKDIMENSIONNOTVALID					: UINT := 2197; (* Dimensioni Pacco presente su Ribaltino non Valide *)
	ErrPALLETCODENOTFOUND						: UINT := 2198; (* Codice pallet non trovato *)
	ErrLAYERCODENOTFOUND						: UINT := 2199; (* Codice layer non trovato *)
	ErrPACKCODENOTFOUND							: UINT := 3000; (* Codice Pacco non trovato in nessuna Formatura *)
	
	(******************************************************************************************************************************************)
	(* Modules Errors *)
	(******************************************************************************************************************************************)
	(* Palletizer *)
	ErrTOADDAXIS								: UINT := 2200; (* Timeout Add Axis *)
	ErrTOUNGROUPALLAXIS							: UINT := 2201; (* Timeout Ungroup All Axis *)
	ErrTOENABLEGROUP							: UINT := 2202; (* Timeout Enable Group *)
	ErrTODISABLEGROUP							: UINT := 2203; (* Timeout Disable Group *)
	ErrTOSTOPGROUP								: UINT := 2004;
	ErrTOUCHEMERGENCY							: UINT := 2205; (* Tastatori Pinza *)
	ErrLOADLOST									: UINT := 2206; (* Perdita Carico Pinza *)
	ErrYBELTSAFETY								: UINT := 2207; (* Sicurezza cinghia asse Y *)
	ErrZBELTSAFETY								: UINT := 2208; (* Sicurezza cinghia asse Z *)
	ErrCOMUNICAZTRASPORTI						: UINT := 2209; (* Mancanza comunicazione con i trasporti *)
	
	ErrMODULEPALLETIZERROBOT_EVSUCTIONUP_TO		: UINT := 2300; (* Timeout Ventose Alte *)
	ErrMODULEPALLETIZERROBOT_EVSUCTIONDOWN_TO	: UINT := 2301; (* Timeout Ventose Basse *)
	ErrMODULEPALLETIZERROBOT_PICKLAYER_TO		: UINT := 2302;
	ErrMODULEPALLETIZERROBOT_EMPTYLAYERSTACK	: UINT := 2303;
	ErrMODULEPALLETIZERROBOT_EMPTYPALLETSTACK	: UINT := 2304;	
	ErrMODULEPALLETIZERROBOT_PRODUCTONGRIPPER	: UINT := 2305;	(* Presenze di materiale non ammesso nella pinza *)
	ErrTOUCHSENSORNOTFREE						: UINT := 2306;
	ErrPALLETNOTPRESENT							: UINT := 2307; (* Pallet non presente per deposito *)	
	ErrPALLETALREADYPRESENT						: UINT := 2308; (* Pallet già presente *)
		
	ErrQUOTAZ_PACCOFUORIING_ELEVATA				: UINT := 2400; (* La quota calcolata di fuori ingombro con PACCO a bordo supera il valore massimo ammesso dall'asse*)
	ErrQUOTAZ_PALLFUORIING_ELEVATA				: UINT := 2401; (* La quota calcolata di fuori ingombro con PALLET a bordo supera il valore massimo ammesso dall'asse*)
	ErrQUOTAZ_VUOTOFUORIING_ELEVATA				: UINT := 2402; (* La quota calcolata di fuori ingombro A VUOTO a bordo supera il valore massimo ammesso dall'asse*)
	ErrQUOTAZ_FALDAFUORIING_ELEVATA				: UINT := 2403; (* La quota calcolata di fuori ingombro con FALDA a bordo supera il valore massimo ammesso dall'asse*)

	ErrPRESENZA_MATERIALE_SUPINZA_CICLO_RIPOSO		: UINT := 2410; (* Presnza materiale non previsto in fase di inizializzazione del ciclo di riposo *)
	ErrPRESENZA_MATERIALE_SUPINZA_CICLO_PRELPALL	: UINT := 2411; (* Presnza materiale non previsto in fase di inizializzazione del ciclo di Prelievo Pallet *)
	ErrPRESENZA_MATERIALE_SUPINZA_CICLO_PRELFALDA	: UINT := 2412; (* Presnza materiale non previsto in fase di inizializzazione del ciclo di Prelievo Falda *)
	ErrPRESENZA_MATERIALE_SUPINZA_CICLO_PRELPACCO	: UINT := 2413; (* Presnza materiale non previsto in fase di inizializzazione del ciclo di Prelievo Pacco *)
	
	ErroreMANCATO_RESET_MISSIONI					: UINT := 2420; (* Errore dovuto al mancato reset della missione, avviene dopo un errore se non è stata aperta la pinza per resettare il tutto *)
	
	ErroreACT_POSX_NONCONFORME   					: UINT := 2421; (* La posizione attuale dell'asse X non rientra nei limiti imposti dal WorkSpace *)
	ErroreACT_POSY_NONCONFORME   					: UINT := 2422; (* La posizione attuale dell'asse Y non rientra nei limiti imposti dal WorkSpace *)
	ErroreACT_POSZ_NONCONFORME   					: UINT := 2423; (* La posizione attuale dell'asse X non rientra nei limiti imposti dal WorkSpace *)
	ErroreACT_POSJ_NONCONFORME   					: UINT := 2424; (* La posizione attuale dell'asse J non rientra nei limiti imposti dal WorkSpace *)	
	
	ErrQUOTEDEPOSITO_NONCONFORMI					: uint := 2425; (* La posizione di deposito pacco non rientra all'interno dell'area di lavoro *)					
	
	ErrMALFUNZIONAMENTOTASTATORI_DURANTETASTEGGIO	: UINT := 2430; (* Durante la risalita dal tasteggio i sensori non leggono correttamente.. verificare l'integrità/il posizionamento dei sensori sulla pinza*)
	
	
	ErrGENERICO : UINT := 9999;

	ErrCYLINDER 						: UINT := 14; (* Cyclinder TF Error *)

	(* Nella gestione errori utilizzare il livello base+l'errore dato dalla libreria*)
	ErrBASEOVEM							: UINT := 30000;
	
	ErrMalfunzionamentoSensoriPresenzaPinza : UINT := 2500;(* Errore di presenza materiale sulla pinza in fase di prelievo, verificare i sensori: FTC/Ovem*)	

	ErrPOSIZIONE_PINZA_ANOMALA				: UINT := 2426; (* La posizione della pionza è anomale per il tipo di movimento che deve svolgere la macchina, blocco per evitare collisioni *)					
	ErrMANCATO_PRELIEVO 					: UINT := 2501;(* Errore di mancato prelievo del pezzo *)	
	
	ErrCOLLISIONE_PINZA						: UINT := 2427; (* La posizione della pinza è anomale per il tipo di movimento che deve svolgere la macchina, blocco per evitare collisioni *)					
	ErrEsMisionSinDimesionPieza				: UINT := 6900 ; (*La Estructura mision no tiene las dimensiones de la pinza*)
END_VAR

// ---- Global Variables/TFCmdStates.TcGVL
{attribute 'Tc2GvlVarNames'}
VAR_GLOBAL CONSTANT
	
	(* Command *)
	CmdPICK 								: UINT := 2000;
	CmdPLACE			 					: UINT := 2100;
	CmdSWAP			 						: UINT := 2200;
	CmdMAINTENANCE 							: UINT := 2300;
	CmdLEARN								: UINT := 2400;

	CmdMOVETOPOS							: UINT := 2600;		// Muovi a posizione data
	CmdMOVEJOG								: UINT := 2700;		// Movimento in jog..Per tasteggio
	CmdTASTEGGIO							: UINT := 2800;		//Comando per tasteggio con FTC per penza basculante

	CmdHALT									: UINT := 2900;

	CmdMOVE		 							: UINT := 3000;
	CmdCYCLEPALLET							: UINT := 4100;
	CmdCYCLELAYER							: UINT := 4200;
	CmdRAISE								: UINT := 4300;
	CmdLOOPPLACE							: UINT := 4400;
	
	CmdPRINT								: UINT := 4500;
	
	CmdCICLORIPOSO							: UINT := 5000;
	
	CmdLOADSEMPLICE							: UINT := 6000;
	CmdUNLOADSEMPLICE						: UINT := 7000;
		
	CmdCHECKPRESENCE						: UINT := 1100; //Comando che valuta la presenza di un oggetto depositato, il suo end arriva se una FTC è intercettatta
	StateCHECKPRESENCE_RUN 					: UINT := 1100; 
	StateCHECKPRESENCE_END 					: UINT := 1199;
	
	


	(* State *)
	StatePICK_RUN 							: UINT := 2000;
	StatePICK_END 							: UINT := 2099;
	StatePLACE_RUN 							: UINT := 2100;
	StatePLACE_END 							: UINT := 2199;
	StateSWAP_RUN 							: UINT := 2200;
	StateSWAP_END 							: UINT := 2299;
	StateMAINTENANCE_RUN 					: UINT := 2300;
	StateMAINTENANCE_END 					: UINT := 2399;
	StateLEARN_RUN							: UINT := 2400;
	StateLEARN_END							: UINT := 2499;

	StateMOVETOPOS_RUN						: UINT := 2600;
	StateMOVETOPOS_END						: UINT := 2699;
	
	StateMOVEJOG_RUN						: UINT := 2700;
	StateMOVEJOG_END						: UINT := 2799;

	StateTASTEGGIO_RUN						: UINT := 2800;
	StateTASTEGGIO_END						: UINT := 2899;

	StateHALT_RUN							: UINT := 2800;
	StateHALT_END							: UINT := 2899;

	StateMOVE_RUN 							: UINT := 3000;
	StateMOVE_END 							: UINT := 3099;
	
	StateCYCLEPALLET_RUN 					: UINT := 4100;
	StateCYCLEPALLET_END 					: UINT := 4199;
	StateCYCLELAYER_RUN 					: UINT := 4200;
	StateCYCLELAYER_END 					: UINT := 4299;
	StateRAISE_RUN							: UINT := 4300;
	StateRAISE_END							: UINT := 4399;
	StateLOOPPLACE_RUN						: UINT := 4400;
	StateLOOPPLACE_END						: UINT := 4499;
	
	StatePRINT_RUN							: UINT := 4500;
	StatePRINT_END							: UINT := 4599;
	
	StateCICLORIPOSO_RUN					: UINT := 4600;
	StateCICLORIPOSO_END					: UINT := 4699;
END_VAR

// ---- Global Variables/TFUpsVariables.TcGVL
{attribute 'Tc2GvlVarNames'}
VAR_GLOBAL
	
	(* UPS *)
	fbUPS			: FB_S_UPS_CX51x0;			(* UPS-FB instance *)
					(* Default Values of FB_S_UPS_CX51x0-Inputs:
						sNetID 			:= '' ==> local netid
						iPLCPort 		:= AMSPORT_R0_PLC_RTS1 ==> 801 = 1st Runtime System
						iUPSPort		:= 16#588 ==> Port for reading Power State of UPS
						tTimeout 		:= DEFAULT_ADS_TIMEOUT ==> 5S
						eUpsMode 		:= eSUPS_WrPersistData_Shutdown ==> writing persistent data + shutdown
						ePersistentMode := SPDM_2PASS ==> All data is from same plc cycle, cycletime exceeds possible. Plc stops with the shutdown, a few cycles after writing persistent data. 
						tRecoverTime 	:= T#10s ==> 10s power to recover from short power failure before eSUPS_PowerOK is reported (in mode eSUPS_WrPersistData_NoShutdown/eSUPS_CheckPowerStatus)
					*)
	eUpsMode		: E_S_UPS_Mode	:= eSUPS_WrPersistData_Shutdown; (* UPS mode (writing persistent data + shutdown) *)

END_VAR

VAR_GLOBAL PERSISTENT
	
	iPowerCounter			: UDINT;			(* Power Counter *)
	iPowerFailureCounter	: UDINT;			(* Power Failures Counter *)
	
END_VAR

// ---- Global Variables/TFVariable/TF_CambioProduzione.TcGVL
{attribute 'Tc2GvlVarNames'}
VAR_GLOBAL PERSISTENT
	// Dati in scambio - EAP
	DatiCambioProduzione_IN AT %I* : DATI_CAMBIO_PRODUZIONE_GENERAL;
	StatoElementoPrecedente AT %I* : STATO_ELEMENTO_GENERAL;
	DatiCambioProduzione_OUT AT %Q* : DATI_CAMBIO_PRODUZIONE_GENERAL;
	StatoElementoASuccessivo AT %Q* : STATO_ELEMENTO_GENERAL;
	
	
	// Dati da supervisione
	RicettaCambioProd : DATI_RICETTA_CONDIVISA;
	
	CambioProd : TFCambioProduzioneLineaGENERAL;
	
	RichiestaCambiodaHMI : BOOL;
	ResetAllarmiModulo : BOOL;
	DatiCambioDaRete : BOOL;						// Stabilisce se le informazioni per eseguire il cambio prod vengono prelevate dalla rete o dal supervisore
	
	ConfigurazioneModulo : CONFIGURAZIONE_ELEMENTO;
	ComandiModulo : COMANDI;
	InputModulo : INPUT_GENERAL;
	ComunicazioneModulo : COMUNICAZIONE_GENERAL;
	
	CambioEseguito_Macchina : BOOL;					// Segnalazione da macchina di cambio produzione eseguito
	CambioRichiesto_Macchina : BOOL;				// Richiesta da modulo a macchina per effettura cambio produzione
	
	AbilitaCambioGlobale : BOOL;
END_VAR

// ---- Global Variables/TO_HMI.TcGVL
{attribute 'Tc2GvlVarNames'}
VAR_GLOBAL	
	AutoMan									: BOOL;

	HMI_Stato_Postazione : ARRAY[1..MAXAREA] OF StatoPostazioneHMI;

	//Stato sicurezze
	HMI_Status_FungiPal_OK 			: BOOL; //Stato funghi pallettizzatore
	HMI_Status_FungoGenerale_OK 	: BOOL; //Stato funghi generali
	HMI_Status_Funghi_OK			: BOOL; //Cumulativo Funghi
		    
	HMI_Status_BarrierDXPal_OK 			: BOOL; //Stato barriera DX
	HMI_Status_BarrierSXPal_OK 			: BOOL; //Stato barriera SX
	HMI_Status_BarrierCentroDXPal_OK	: BOOL; //Stato barriera CENTRO-DX
	HMI_Status_BarrierCentroSXPal_OK	: BOOL; //Stato barriera CENTRO-SX
	HMI_Status_StateBarrierKarv_OK    	: BOOL; //Stato barriera KARV
	HMI_Status_BarrieraPall_OK			: BOOL; //Stato COMULATIVO BARRIERE	
	
	HMI_WorkAreaProductionList : ARRAY [1..MAXAREA] OF TFMachinePalletizer_ListaProduzione_WAM_HMI;//Variabile per visuallizzare su HMI lo stato della lista di produzione
	
	// VARIABILI PER VISUALIZZAZIONE I/O SU HMI PREMIUM
	HMI_AP200_2 : ARRAY[1..16] OF BOOL;
	HMI_AP200_3 : ARRAY[1..4] OF BOOL;
	HMI_AP200_4 : ARRAY[1..4] OF BOOL;
	HMI_AP200_5 : ARRAY[1..16] OF BOOL;
	HMI_AP200_6	: ARRAY[1..4] OF BOOL;
	HMI_AP200_7	: ARRAY[1..4] OF BOOL;
	HMI_AP200_8 : ARRAY[1..16] OF BOOL;
	HMI_AP200_9	: ARRAY[1..4] OF BOOL;
	HMI_AP200_10: ARRAY[1..4] OF BOOL;
	HMI_AP201_2	: ARRAY[1..4] OF BOOL;
	HMI_AP201_4 : ARRAY[1..16] OF BOOL;
	HMI_AP201_5	: ARRAY[1..4] OF BOOL;
	HMI_AP201_6 : ARRAY[1..16] OF BOOL;
	HMI_AP201_3 : ARRAY[1..16] OF BOOL;
	HMI_AP202_2	: ARRAY[1..4] OF BOOL;
	HMI_AP202_3	: ARRAY[1..4] OF BOOL;
	HMI_AP202_5	: ARRAY[1..4] OF BOOL;
	HMI_AP202_6	: ARRAY[1..4] OF BOOL;
	
	//CIABATTA 515
	HMI_DepressioneOVEM_SX1 	: REAL; //Valore porta 1
	//
	HMI_LetturaFTCPinza0_1 		: REAL; //Valore porta 3
	HMI_LetturaFTCPinza180_1	: REAL; //Valore porta 4
	HMI_DepressioneOVEM_SX2 	: REAL; //Valore porta 5
	//CIABATTA 516	
	HMI_DepressioneOVEM_DX1 	: REAL; //Valore porta 1
	HMI_DepressioneOVEM_DX2 	: REAL; //Valore porta 2
	HMI_LetturaFTCPinza0_2		: REAL; //Valore porta 3
	HMI_LetturaFTCPinza180_2 	: REAL; //Valore porta 4
	HMI_K516_51 				: BOOL;//Valore porta 5
	HMI_K516_52 				: BOOL;//Valore porta 5
	HMI_K516_61 				: BOOL;//Valore porta 6 pin 4
	HMI_K516_62 				: BOOL;//Valore porta 6 pin 2
	HMI_K516_71 				: BOOL;//Valore porta 7 pin 4
	HMI_K516_72 				: BOOL;//Valore porta 7 pin 2
	HMI_K516_81 				: BOOL;//Valore porta 8 pin 4
	HMI_K516_82 				: BOOL;//Valore porta 8 pin 2
	//CIABATTA 517	
	HMI_K517_11  				: BOOL;//Valore porta 1
	HMI_K517_12  				: BOOL;//Valore porta 1
	HMI_K517_21  				: BOOL;//Valore porta 2
	HMI_K517_22  				: BOOL;//Valore porta 2
	HMI_K517_31  				: BOOL;//Valore porta 3
	HMI_K517_32  				: BOOL;//Valore porta 3
	HMI_K517_41  				: BOOL;//Valore porta 4
	HMI_K517_42  				: BOOL;//Valore porta 4
	HMI_K517_51 				: BOOL;//Valore porta 5
	HMI_K517_52 				: BOOL;//Valore porta 5
	HMI_K517_61 				: BOOL;//Valore porta 6 pin 4
	HMI_K517_62 				: BOOL;//Valore porta 6 pin 2
	HMI_K517_71 				: BOOL;//Valore porta 7 pin 4
	HMI_K517_72 				: BOOL;//Valore porta 7 pin 2
	HMI_K517_81 				: BOOL;//Valore porta 8 pin 4
	HMI_K517_82 				: BOOL;//Valore porta 8 pin 2

	
	Control1: INT;
END_VAR

// ---- POUs/TFPrograms/TFMachinePalletizerMain.TcPOU
PROGRAM TFMachinePalletizerMain
VAR
	ManCmdXHomeTRIG 			: BOOL;
	ManCmdYHomeTRIG 			: BOOL;
	ManCmdZHomeTRIG 			: BOOL;
	ManCmdJHomeTRIG 			: BOOL;
	ManCmdKHomeTRIG 			: BOOL;
	ManCmdGeneralHomeTRIG 		: BOOL;
	
	Formacion_bandelCalOk		:ARRAY [1..3] OF BOOL ;
	Formacion_FrameCalOk		:ARRAY [1..3] OF BOOL ;
	Formacion_De_listaOk		:ARRAY [1..3] OF BOOL ;
	 

	i : UINT;
	k : UINT;
	j : UINT;
	TEST_ENABLE 		: BOOL:= FALSE;
	POTENZA_TEST_ENABLE : BOOL:= FALSE;
	TestSenzaHw 		: BOOL;
	DriveNeedReset 		: BOOL := TRUE;
	first 				: BOOL;
	InitWAZone 			: BOOL;
	EmergenzeOK_Simulazione : BOOL;
	SimulaArrayPacchi 		: BOOL;
	iLgv 					: UINT;//Indice per aggiornare dati verso bridge navette
	iLgvPack 				: UINT;//Indice per aggiornare pacchi formature dati verso bridge navette
	iLgvPackP				: UINT;
	iLgvPackN 				: UINT;
	AggioraDatiLgv			: UINT;
	Post 					: UINT;
	CmdJogNeg_X 			: BOOL;
	CmdJogPos_X 			: BOOL;
	PowerEnableAssi 		: BOOL; //Presneza marcia e abilitazione power assi
	Auto_GENERAL			: INT;
	TotalePacchiParziali	: DWORD;
	TimerConsensoValle 		: REAL;
	TimerAutomaticoValle 	: REAL;
	GestionePickPoint 		: TFPalletizerGestione_PickPoint_Rulliere;
	CalcolaFormaturaTrig 	: BOOL;
	icode 					: UINT;
	icode2 					: UINT;
	iform 					: UINT;
	DisablePowerPerConfig 	: BOOL;
	AggiuntaPalletManuale 			: TFAggiuntaSupportoManuale;
	FiltroFTCPalletPerManuale		: ARRAY[1..MAXAREA] OF Signal_Filter;
	TFCalcolaNumeroPostazioneDXSX 	: TFCalcolaNumeroPostazioneDXSX;
	postest 						: REAL;
	iformaturatest 					: UINT := 2;
	fbGetCurTaskIdx  				: GETCURTASKINDEX;
	
	idxForm : uint;
	CalcolaFormaturaTrig2 : BOOL;
	CalcolaFormingRT : ARRAY[1..3] OF BOOL;
	CalcolaFormingRT2 : ARRAY[1..3] OF BOOL;
	IdxLista : UINT;
	Iforstart : UINT;
	Iforend : UINT;
	TimerAggancioBloccoDicurezza 	: Tc2_Standard.TOF;
	InPosPx: INT;
	Prueva: BOOL;
	MissionClr : POINTER TO TFMachinePalletizer_Mission;
	
	TraiettoriaClr : POINTER TO TFTraiettoria;
	jj: UINT;
	ClrEstructura: POINTER TO ARRAY [1..MAXPALLET] OF e_Tipo_Pallet;
	// Variable para rellenar la estrctura con las dimensiones de la pieza
	InPiezasPos: UINT;
	// Variable pafa Calcular las formaciones
	CalFor: UINT;
	// Recorre los casos para crear la formacion
	CrearFormacion: UINT;
	uu: UINT;
	
	HH: INT;
	Hhbilita_quitar: BOOL;
	ja: UINT;
	
	pr1: UINT;
	pr2: UINT;
	P_ladoA: UINT;
	P_ladoB: UINT;
	LadoRegistar: UINT;
	CooCavallete: INT;
	DD: UINT;
	HolaCabron :INT ;
END_VAR

_01_Init();
_02_LeggiInput();
_03_Modules();
_04_Comunicazione();
_05_ManualCmds();
_06_ScriviOutput();
_07_ScriviStatus();
//_08_DataLogger_ACT();
//_09_CalcolaFormatura();
_10_PackModifier();
IF NOT HabilitacionFormacionNueva THEN 
	_11_CalcolaListaProduzione();
ELSE
	_11_CalcolaListaProduzioneNew();	
END_IF

//##
Test_Variabili();
//##

ACTION _01_Init:
//Al primo giro di PLC inizializzo le variabili che mi servono
fbGetCurTaskIdx();
IF _TaskInfo[fbGetCurTaskIdx.index].FirstCycle THEN
	TimeBase := UDINT_TO_REAL(_TaskInfo[fbGetCurTaskIdx.index].CycleTime/10000);//Valorizzazione del tempo ciclo del PLC
	LOCAL_AmsNetId := F_CreateAmsNetId(AmsNetId);
	
	HMI_NumeroPezziPresentiPostazione[i] := WorkAreaState[i].P-1; 	
	
	OffsetDistacco.Lastra.Z := 30;
	OffsetDistacco.Lastra.Y := 30;
	
	OffsetSicurezza.Y.Avuoto := 200; //Canada 300
	OffsetSicurezza.Y.Carico := 200; //canada 300
	
	OffsetSicurezza.Z.Avuoto := 200;
	OffsetSicurezza.Z.Carico := 350;
	IF Habilito_Pos_j_Fc THEN 
		HMI_AbilitaPosJPrelConFTC := TRUE;
	ELSE
		HMI_AbilitaPosJPrelConFTC := FALSE;
	END_IF
		
	
END_IF


IF MachinePalletizerInitVariables THEN
	MachinePalletizerInitVariables := FALSE;
	NUMERO_MACCHINA := 1;
	(***********************************************************************************************************************************************************************************)
	(***********************************************************************************************************************************************************************************)
	VERSO_PALLETTIZZATORE 			 	:= PALLETTIZZATORE_SX; 		//Verso Pallettizzatore: stabilito guardando il pallettizzatore con la linea alle spalle
	TIPO_MAGAZZINO_FALDE  			 	:= MAGAZZINO_FALDE_IN_WA; 	//Identifica il tipo di magazzino falde: MAGAZZINO_FALDE_CENTRO_FISSO = LA Y DI PRELIEVO RIMANE COSTANTE PER OGNI FORMATO,MAGAZZINO_FALDE_CENTRO_VARIABILE=LA Y DI PRELIEVO SI ADATTA AL FORMATO DELLA FALDA
	RIFERIMENTO_POSTAZIONE_WA			:= e_RiferimentoPostazione.CENTRALE;
	ASSE_DISPOSIZIONE_POSTAZIONI		:= e_Disposizione_Postazioni.LUNGO_X;
	TIPOLOGIA_FUNZIONAMENTO_MACCHINA	:= FUNZIONAMENTO_PICKING;

	ORDINE_DISPOSIZIONE_POSTAZIONI		:= CRESCENTE;
	
	OFFSET_POSTAZIONE_LEGNO 	:= 1330;// 1200 + 150 anatolia EEUU Offset filo fisso per legni rispetto al filo del bundle che è la quota di riferimento della WORKAREA lungo Y
	OFFSET_POSTAZIONE_TELAIO 	:= 3415 ; //Hay que poner 3125 hay una diferencia 290 sobre la medida real que es 3415//Offset filo fisso per TELAI rispetto al filo del bundle che è la quota di riferimento della WORKAREA lungo Y
	
	INGOMBRO_RISCONTRO_BUNDLE := 100;
	
	MAXAREAPRESENT := 8; //Numeor di postazioni effettivamente presenti in macchina
	(***********************************************************************************************************************************************************************************)
	(* Postazioni *)
	(***********************************************************************************************************************************************************************************)
	NumPostazioneDeposito 			:= 1;// Numero della postazione di deposito materiale
	NumPostazioneSuRulliera			:= 1;// Numero della postazione di deposito materiale su rulliera: se ho pal picking!!	
	NumPostazioneFALDE 				:= 10; //Numero postazione dedicata alle falde
	NumPostazioneDiPareggiatura 	:= 10; //Numero Postazione dedicata alla pareggiatura
	NumPostazioneBundle 			:= 11; //Numero Postazione dedicata al bundle
	AngoloInclinazioneBundle 		:= 7; //Angolo di inclinazione del bundle

	AngoloInclinazioneTavolaPareggiatura := 7;//173; //Gradi di inclinazione della Tavola di pareggiatura
	(***********************************************************************************************************************************************************************************)
	(* Spazio di lavoro *)
	(***********************************************************************************************************************************************************************************)
	WorkSpace.X := 33345;
	WorkSpace.Y := 3300; // 3120
	WorkSpace.Z := 1730;
	(***********************************************************************************************************************************************************************************)
	(* Quote Punto di Prelievo 1 *)
	(***********************************************************************************************************************************************************************************)
	WorkPickPoint[1].X := 155;
	WorkPickPoint[1].Y := 2800;
	WorkPickPoint[1].Z := 0;
	WorkPickPoint[1].J := 90;
	WorkPickPoint[1].ZRaise := 0;
	WorkPickPoint[1].Enable := 0;
	WorkPickPoint[1].Tipologia := RULLIERA;

	(* Dimensioni fisiche Punto di Prelievo *)
	WorkPickPointDimension[1].Xdim := 0;
	WorkPickPointDimension[1].Ydim := 0;
	WorkPickPointDimension[1].Zdim := 0;
	
	(* Ingombri *)
	WorkFootprint[1].X := 5385;
	WorkFootprint[1].Y := 15;
	WorkFootprint[1].Z := 0;//10;
	WorkFootprint[1].XDim := 20;
	WorkFootprint[1].YDim := 1000;
	WorkFootprint[1].ZDim := 500;//900;
	
	WorkFootprint[2].X := 6669;
	WorkFootprint[2].Y := 15;
	WorkFootprint[2].Z := 0;//10;
	WorkFootprint[2].XDim := 20;
	WorkFootprint[2].YDim := 1000;
	WorkFootprint[2].ZDim := 900;//900;
	
	WorkFootprint[3].X := 7184;
	WorkFootprint[3].Y := 15;
	WorkFootprint[3].Z := 0;//10;
	WorkFootprint[3].XDim := 20; //0;
	WorkFootprint[3].YDim := 1700; //0;
	WorkFootprint[3].ZDim := 500; //0;
	
	WorkFootprint[4].X := 8100;
	WorkFootprint[4].Y := 15;
	WorkFootprint[4].Z := 0; //10;
	WorkFootprint[4].XDim := 20;//0;
	WorkFootprint[4].YDim := 1700;//0;
	WorkFootprint[4].ZDim := 500;//0;
	
	CASE VERSO_PALLETTIZZATORE OF
		PALLETTIZZATORE_DX:
			(* Colonna SX *)				//valori online
			WorkFootprint[5].X := 5020;
			WorkFootprint[5].Y := 3356;		//0
			WorkFootprint[5].Z := 300; 
			WorkFootprint[5].XDim := 300;
			WorkFootprint[5].YDim := 0;
			WorkFootprint[5].ZDim := 0;
			
			(* Colonna DX *)
			WorkFootprint[6].X := 5020;
			WorkFootprint[6].Y := 0;		//3360
			WorkFootprint[6].Z := 0; 		//300
			WorkFootprint[6].XDim := 300;
			WorkFootprint[6].YDim := 0;
			WorkFootprint[6].ZDim := 0;
		
		PALLETTIZZATORE_SX:
			(* Colonna SX *)
			WorkFootprint[5].X := 5020;
			WorkFootprint[5].Y := 0;
			WorkFootprint[5].Z := 300; 
			WorkFootprint[5].XDim := 300;
			WorkFootprint[5].YDim := 0;
			WorkFootprint[5].ZDim := 0;
			
			(* Colonna DX *)
			WorkFootprint[6].X := 5020;
			WorkFootprint[6].Y := 3050;
			WorkFootprint[6].Z := 0; 		//300
			WorkFootprint[6].XDim := 300;
			WorkFootprint[6].YDim := 0;
			WorkFootprint[6].ZDim := 0;
			
	END_CASE
	
	(* Postazioni *)
	WorkArea[1].Enable := 1;
	WorkArea[1].Typology := TYPOLOGY_PALLET;
	WorkArea[1].X := 2118; // 2128;
	WorkArea[1].Y := 745; //877;
	WorkArea[1].Z := 0;
	WorkAreaState[1].H := 0;
	WorkAreaState[1].HPL := 0;

	WorkArea[2].Enable := 1;
	WorkArea[2].Typology := TYPOLOGY_PALLET;
	WorkArea[2].X := 6210; //6270;
	WorkArea[2].Y := 745; //877;
	WorkArea[2].Z := 0;
	WorkAreaState[2].H := 0;
	WorkAreaState[2].HPL := 0;

	WorkArea[3].Enable := 1;
	WorkArea[3].Typology := TYPOLOGY_PALLET;
	WorkArea[3].X := 10699; //10744;
	WorkArea[3].Y := 745; //877;
	WorkArea[3].Z := 0;//595;
	WorkAreaState[3].H := 0;
	WorkAreaState[3].HPL := 0;

	WorkArea[4].Enable := 1;
	WorkArea[4].Typology := TYPOLOGY_PALLET;
	WorkArea[4].X := 14789; //14844;
	WorkArea[4].Y := 745; //877;
	WorkArea[4].Z := 0;
	WorkAreaState[3].H := 0;
	WorkAreaState[3].HPL := 0;

	WorkArea[5].Enable := 0;
	WorkArea[5].Typology := TYPOLOGY_PALLET;
	WorkArea[5].X := 19189; //18944;
	WorkArea[5].Y := 745; //877; //755;
	WorkArea[5].Z := 0;
	WorkAreaState[5].H := 0;
	WorkAreaState[5].HPL := 0;

	WorkArea[6].Enable := 0;
	WorkArea[6].Typology := TYPOLOGY_PALLET;
	WorkArea[6].X := 23303; //23418;
	WorkArea[6].Y := 745; //877;//755;
	WorkArea[6].Z := 0;
	WorkAreaState[6].H := 0;
	WorkAreaState[6].HPL := 0;
	
	WorkArea[7].Enable := 1;
	WorkArea[7].Typology := TYPOLOGY_PALLET;
	WorkArea[7].X := 27792; //27892;
	WorkArea[7].Y := 745; //877;
	WorkArea[7].Z := 0;
	WorkAreaState[7].H := 0;
	WorkAreaState[7].HPL := 0;

	WorkArea[8].Enable := 0;
	WorkArea[8].Typology := TYPOLOGY_PALLET;
	WorkArea[8].X := 31872; //31992;
	WorkArea[8].Y := 745; //877;
	WorkArea[8].Z := 0;
	WorkAreaState[8].H := 0;
	WorkAreaState[8].HPL := 0;
	
		
	WorkAreaState[1].State := 0;
	WorkAreaState[1].F := -1;
	WorkAreaState[1].P := -1;
	
	WorkAreaState[2].State := 0;
	WorkAreaState[2].F := -1;
	WorkAreaState[2].P := -1;
	
	WorkAreaState[3].State := 0;
	WorkAreaState[3].F := -1;
	WorkAreaState[3].P := -1;

	WorkAreaState[4].State := 0;
	WorkAreaState[4].F := -1;
	WorkAreaState[4].P := -1;

	WorkAreaState[5].State := 0;
	WorkAreaState[6].State := 0;
	WorkAreaState[7].State := 0;
	WorkAreaState[8].State := 0;


	(* Pallet *)
	Pallet[1].XDim := 800;
	Pallet[1].YDim := 1200;
	Pallet[1].ZDim := 125;
	(* Falde *)
	Layer[1].XDim := 800;
	Layer[1].YDim := 1200;
	Layer[1].ZDim := 2.8;
		
	TCPParameter.X := 0;
	TCPParameter.Y := 0;
	TCPParameter.Z := 112;
	
	PreviousStackWA	:= 1;
	
	HMI_OverideDinamico.NTrasportiOccupati[1] := 7;
	HMI_OverideDinamico.Override[1] := 100;
	HMI_OverideDinamico.NTrasportiOccupati[2] := 5;
	HMI_OverideDinamico.Override[2] := 80;
	HMI_OverideDinamico.NTrasportiOccupati[3] := 3;
	HMI_OverideDinamico.Override[3] := 60;
	HMI_OverideDinamico.NTrasportiOccupati[4] := 1;
	HMI_OverideDinamico.Override[4] := 40;
	
	HMI_AxisOverride.Auto := 50;
	HMI_AxisOverride.Jog := 50;
	HMI_AxisOverride.Layer := 50;
	HMI_AxisOverride.Pallet := 50;
	HMI_AxisOverride.Pack := 50;
	HMI_AxisOverride.PickRip := 50;
	
	Dimensioni_Pinza.Lunghezza 			:= 2410; // Comprese le ventose ??? (ex1650) ;
	Dimensioni_Pinza.Larghezza 			:= 930;  // Comprese le ventose ??? (ex780);
	Dimensioni_Pinza.Spessore 			:= 300;  // Compresa ventosa
	Dimensioni_Pinza.DimTraveVerticale 	:= 150; 

	OffsetDistacco.Lastra.Y := 30;//5;
	OffsetDistacco.Lastra.Z := 30;

	(* Variabili per posizione di riposo*)
	X_Riposo	:= WorkArea[1].X;
	Y_Riposo	:= WorkArea[1].Y;
	Z_Riposo	:= 1826;
	J_Riposo	:= 90;

END_IF

IF MachinePalletizerInitDone THEN	
	MachinePalletizerInitDone := FALSE;

	//LearnParameters.Velocity := AxisPar.Z.MaxVelocity * 0.08;

	AxisNominalPar_X.ReferenceVelocity := 2600;
	AxisNominalPar_X.MaximumAcceleration := 2000;//2188.23;
	AxisNominalPar_X.MaximumDeceleration := 2000;//2188.23;
	AxisNominalPar_X.DefaultJerk := 6650.4799999999996;
	AxisNominalPar_X.DefaultTorque := 0;
	
	AxisNominalPar_Y.ReferenceVelocity := 1800;
	AxisNominalPar_Y.MaximumAcceleration := 1000.0;
	AxisNominalPar_Y.MaximumDeceleration := 1000.0;
	AxisNominalPar_Y.DefaultJerk := 7920.5100000000002;
	AxisNominalPar_Y.DefaultTorque := 0;

	AxisNominalPar_Z.ReferenceVelocity := 520.0;
	AxisNominalPar_Z.MaximumAcceleration := 2500;
	AxisNominalPar_Z.MaximumDeceleration := 2500;
	AxisNominalPar_Z.DefaultJerk := 11221;
	AxisNominalPar_Z.DefaultTorque := 0;

	AxisNominalPar_J.ReferenceVelocity := 100;
	AxisNominalPar_J.MaximumAcceleration := 300;
	AxisNominalPar_J.MaximumDeceleration := 300;
	AxisNominalPar_J.DefaultJerk := 20000;
	AxisNominalPar_J.DefaultTorque := 0;
	(*
	AxisNominalPar_K.ReferenceVelocity := 224;
	AxisNominalPar_K.MaximumAcceleration := 5000;
	AxisNominalPar_K.MaximumDeceleration := 5000;
	AxisNominalPar_K.DefaultJerk := 50000;
	AxisNominalPar_K.DefaultTorque := 100;	
	*)
	AxisPar_X.Acc := AxisNominalPar_X.MaximumAcceleration;
	AxisPar_X.Dec := AxisNominalPar_X.MaximumDeceleration;
	AxisPar_X.Vel := AxisNominalPar_X.ReferenceVelocity;
	AxisPar_X.MaxAcc := AxisNominalPar_X.MaximumAcceleration;
	AxisPar_X.MaxDec := AxisNominalPar_X.MaximumDeceleration;
	AxisPar_X.MaxVel := AxisNominalPar_X.ReferenceVelocity;
	AxisPar_X.ManFastVel := 15;
	AxisPar_X.ManSlowVel := 1;
	AxisPar_X.JOGAcc := AxisNominalPar_X.MaximumAcceleration;
	AxisPar_X.JOGDec := AxisNominalPar_X.MaximumDeceleration;
	AxisPar_X.Jerk := AxisNominalPar_X.DefaultJerk;
	AxisPar_X.MaxPosition := WorkSpace.X;
	AxisPar_X.HomeDefine := 715.0; (*+700 +15 Anatolia Canada*)
	AxisPar_X.HomePosition := 715; (*700 +15 Anatolia Canada*)
	AxisPar_X.MinPosition := 699;//AxisPar_X.HomeDefine;
	AxisPar_X.HomeVelocity := 40;
	
	CASE VERSO_PALLETTIZZATORE OF
		PALLETTIZZATORE_DX:	
			InvertiComandoJog_X := FALSE;
		
		PALLETTIZZATORE_SX:
			InvertiComandoJog_X := TRUE;
	END_CASE
	
	
	AxisPar_Y.Acc := AxisNominalPar_Y.MaximumAcceleration;
	AxisPar_Y.Dec := AxisNominalPar_Y.MaximumDeceleration;
	AxisPar_Y.Vel := AxisNominalPar_Y.ReferenceVelocity;
	AxisPar_Y.MaxAcc := AxisNominalPar_Y.MaximumAcceleration;
	AxisPar_Y.MaxDec := AxisNominalPar_Y.MaximumDeceleration;
	AxisPar_Y.MaxVel := AxisNominalPar_Y.ReferenceVelocity;
	AxisPar_Y.ManFastVel := 20;
	AxisPar_Y.ManSlowVel := 2;
	AxisPar_Y.JOGAcc := AxisNominalPar_Y.MaximumAcceleration;
	AxisPar_Y.JOGDec := AxisNominalPar_Y.MaximumDeceleration;
	AxisPar_Y.Jerk := AxisNominalPar_Y.DefaultJerk;
	AxisPar_Y.MaxPosition := 3300;
	AxisPar_Y.HomeDefine := 535.0;
	AxisPar_Y.HomePosition := 535.0;
	AxisPar_Y.MinPosition := 534;
	AxisPar_Y.HomeVelocity := 30;
	
	AxisPar_Z.Acc := AxisNominalPar_Z.MaximumAcceleration;
	AxisPar_Z.Dec := AxisNominalPar_Z.MaximumDeceleration;
	AxisPar_Z.Vel := AxisNominalPar_Z.ReferenceVelocity;
	AxisPar_Z.MaxAcc := AxisNominalPar_Z.MaximumAcceleration;
	AxisPar_Z.MaxDec := AxisNominalPar_Z.MaximumDeceleration;
	AxisPar_Z.MaxVel := AxisNominalPar_Z.ReferenceVelocity;
	AxisPar_Z.ManFastVel := 10;
	AxisPar_Z.ManSlowVel := 2;
	AxisPar_Z.JOGAcc := AxisNominalPar_Z.MaximumAcceleration;
	AxisPar_Z.JOGDec := AxisNominalPar_Z.MaximumDeceleration;
	AxisPar_Z.Jerk := AxisNominalPar_Z.DefaultJerk;
	
	AxisPar_Z.MinPosition := 20;
	AxisPar_Z.MaxPosition := 1730;
	AxisPar_Z.HomeDefine :=  1730;
	AxisPar_Z.HomePosition := 1730.0;
	AxisPar_Z.HomeVelocity := 30;
	
	AxisPar_J.Acc := AxisNominalPar_J.MaximumAcceleration;
	AxisPar_J.Dec := AxisNominalPar_J.MaximumDeceleration;
	AxisPar_J.Vel := AxisNominalPar_J.ReferenceVelocity;
	AxisPar_J.MaxAcc := AxisNominalPar_J.MaximumAcceleration;
	AxisPar_J.MaxDec := AxisNominalPar_J.MaximumDeceleration;
	AxisPar_J.MaxVel := AxisNominalPar_J.ReferenceVelocity;
	AxisPar_J.ManFastVel := 10;
	AxisPar_J.ManSlowVel := 2;
	AxisPar_J.JOGAcc := AxisNominalPar_J.MaximumAcceleration;
	AxisPar_J.JOGDec := AxisNominalPar_J.MaximumDeceleration;
	AxisPar_J.Jerk := AxisNominalPar_J.DefaultJerk;
	
	CASE VERSO_PALLETTIZZATORE OF
		PALLETTIZZATORE_DX:	
		
			AxisPar_J.MaxPosition 	:= 181.6;
			AxisPar_J.HomeDefine 	:= 181.6;
			AxisPar_J.HomePosition 	:= 181.6;
			AxisPar_J.MinPosition 	:= -1;
			
		PALLETTIZZATORE_SX:
		
			AxisPar_J.MaxPosition 	:= 181.0;
			AxisPar_J.HomeDefine 	:= -1.0;
			AxisPar_J.HomePosition 	:= -1.0;
			AxisPar_J.MinPosition 	:= -2.0;
	END_CASE	
	
	AxisPar_J.HomeVelocity := 2;
	
	(*
	AxisPar_K.Acc := 500;
	AxisPar_K.Dec := 500;
	AxisPar_K.Vel := 224;
	AxisPar_K.MaxAcc := AxisNominalPar_K.MaximumAcceleration;
	AxisPar_K.MaxDec := AxisNominalPar_K.MaximumDeceleration;
	AxisPar_K.MaxVel := 224;
	AxisPar_K.ManFastVel := 20;
	AxisPar_K.ManSlowVel := 10;
	AxisPar_K.JOGAcc := AxisNominalPar_K.MaximumAcceleration;
	AxisPar_K.JOGDec := AxisNominalPar_K.MaximumDeceleration;
	AxisPar_K.Jerk := AxisNominalPar_K.DefaultJerk;
	AxisPar_K.MinPosition := 584.0;
	AxisPar_K.MaxPosition := 1200.0;
	AxisPar_K.HomeDefine := 1280.0; 
	AxisPar_K.HomePosition := 800.0;
	AxisPar_K.MaxTorque := 100;
	AxisPar_K.HomeVelocity := 10;
	*)
	(* Parametri HOMING *)
	AxisHomingParameters_X.InvertiDirezione := FALSE;
	AxisHomingParameters_X.TipoHoming 		:= HOMING_STANDARD;
	AxisHomingParameters_Y.InvertiDirezione := FALSE;
	AxisHomingParameters_Y.TipoHoming 		:= HOMING_STANDARD;
	AxisHomingParameters_Z.InvertiDirezione := TRUE;
	AxisHomingParameters_Z.TipoHoming 		:= HOMING_STANDARD;
	AxisHomingParameters_J.InvertiDirezione := TRUE;
	AxisHomingParameters_J.TipoHoming 		:= HOMING_STANDARD;

END_IF

IF InitWAZone THEN
	InitWAZone := FALSE;
	WorkAreaZone.Zone[1].Code[1] := 1;
	WorkAreaZone.Zone[1].Code[2] := 2;
	WorkAreaZone.Zone[1].Code[3] := 3;
	WorkAreaZone.Zone[1].Code[4] := 4;
	WorkAreaZone.Zone[1].Code[5] := 5;
	WorkAreaZone.Zone[1].Code[6] := 6;
	WorkAreaZone.Zone[1].Code[7] := 7;
	WorkAreaZone.Zone[1].Code[8] := 8;
	WorkAreaZone.Zone[1].Code[9] := 9;
	WorkAreaZone.Zone[1].Code[10]:= 10;
	WorkAreaZone.Zone[1].WorkArea[1] := 1;
	WorkAreaZone.Zone[1].WorkArea[2] := 2;
	WorkAreaZone.Zone[1].WorkArea[3] := 3;
	WorkAreaZone.Zone[1].WorkArea[4] := 4;
	WorkAreaZone.Zone[1].WorkArea[5] := 5;
	WorkAreaZone.Zone[1].WorkArea[6] := 6;
	WorkAreaZone.Zone[1].WorkArea[7] := 7;
	WorkAreaZone.Zone[1].WorkArea[8] := 8;
	WorkAreaZone.Zone[1].WorkArea[9] := 9;
	WorkAreaZone.Zone[1].WorkArea[10]:= 10;
	(*
	WorkAreaZone.Zone[2].Code[1] := 7;
	WorkAreaZone.Zone[2].Code[2] := 0;
	WorkAreaZone.Zone[2].Code[3] := 0;
	WorkAreaZone.Zone[2].Code[4] := 0;
	WorkAreaZone.Zone[2].Code[5] := 0;
	WorkAreaZone.Zone[2].Code[6] := 0;
	WorkAreaZone.Zone[2].Code[7] := 0;
	WorkAreaZone.Zone[2].Code[8] := 0;
	WorkAreaZone.Zone[2].Code[9] := 0;
	WorkAreaZone.Zone[2].Code[10] := 0;
	WorkAreaZone.Zone[2].WorkArea[1] := 3;
	WorkAreaZone.Zone[2].WorkArea[2] := 10;
	WorkAreaZone.Zone[2].WorkArea[3] := 0;
	WorkAreaZone.Zone[2].WorkArea[4] := 0;
	WorkAreaZone.Zone[2].WorkArea[5] := 0;
	WorkAreaZone.Zone[2].WorkArea[6] := 0;
	WorkAreaZone.Zone[2].WorkArea[7] := 0;
	WorkAreaZone.Zone[2].WorkArea[8] := 0;
	WorkAreaZone.Zone[2].WorkArea[9] := 0;
	WorkAreaZone.Zone[2].WorkArea[10]:= 0;
	
	WorkAreaZone.Zone[3].Code[1] := 9;
	WorkAreaZone.Zone[3].Code[2] := 0;
	WorkAreaZone.Zone[3].Code[3] := 0;
	WorkAreaZone.Zone[3].Code[4] := 0;
	WorkAreaZone.Zone[3].Code[5] := 0;
	WorkAreaZone.Zone[3].Code[6] := 0;
	WorkAreaZone.Zone[3].Code[7] := 0;
	WorkAreaZone.Zone[3].Code[8] := 0;
	WorkAreaZone.Zone[3].Code[9] := 0;
	WorkAreaZone.Zone[3].Code[10] := 0;
	WorkAreaZone.Zone[3].WorkArea[1] := 2;
	WorkAreaZone.Zone[3].WorkArea[2] := 10;
	WorkAreaZone.Zone[3].WorkArea[3] := 0;
	WorkAreaZone.Zone[3].WorkArea[4] := 0;
	WorkAreaZone.Zone[3].WorkArea[5] := 0;
	WorkAreaZone.Zone[3].WorkArea[6] := 0;
	WorkAreaZone.Zone[3].WorkArea[7] := 0;
	WorkAreaZone.Zone[3].WorkArea[8] := 0;
	WorkAreaZone.Zone[3].WorkArea[9] := 0;
	WorkAreaZone.Zone[3].WorkArea[10]:= 0;*)

END_IF
END_ACTION

ACTION _02_LeggiInput:
(* J17 *)
//I_TastoreCartone1 := I_K517[3].0;
//I_TastoreCartone2 := I_K517[2].0;
//I_ExtraCorsaPinzaSganciata := I_K517[2].6;
//I_PHPresenzaFaldaSX := I_K517[3].4;

I_RotazioneColonnaBloccata 	:= I_K517[2].1; //Ingresso X1.1 pin 4
I_TastatoreBascolante	 	:= I_K517[3].1; //Ingresso X1.1 pin 2
//--
I_PHPresenzaFaldaDX 		:= I_K517[2].2; //Ingresso X1.2 pin 4
//--
//Segnali da Ciabatta
I_TastatorePinza_1 			:= I_K517[2].4;
I_TastatorePinza_2 			:= I_K517[3].4;
//Mod 3_6_2025
I_TastatoreEmergenzaPinza_1 := TRUE;
//I_TastatoreEmergenzaPinza_1 := I_K517[2].5;
I_TastatoreEmergenzaPinza_2 := I_K517[3].5;
//--
I_TastatorePinza_3 			:= I_PortQualCiabattaK516_X05.0;
I_TastatorePinza_4 			:= I_PortQualCiabattaK516_X05.1;
I_TastatoreEmergenzaPinza_3 := I_PortQualCiabattaK516_X06.0;
I_TastatoreEmergenzaPinza_4 := I_PortQualCiabattaK516_X06.1;
//--
I_TastatorePinza_5	:= TRUE;
I_TastatorePinza_6 	:= TRUE;
//--
I_Keyence0_Byte0 	:= I_K515_XO3[0];
I_Keyence0_Byte1 	:= I_K515_XO3[1];
I_Keyence180_Byte0 	:= I_K515_XO4[0];
I_Keyence180_Byte1 	:= I_K515_XO4[1];
//--
I_Keyence0_Byte0_2 	:= I_K516_XO3[0];
I_Keyence0_Byte1_2 	:= I_K516_XO3[1];
I_Keyence180_Byte0_2 := I_K516_XO4[0];
I_Keyence180_Byte1_2 := I_K516_XO4[1];

//Segnali da azionamenti
//originali
//I_ExtraCorsaPositivo_X 	:= I_XDriveDigitalInput.1;
//I_ExtraCorsaNegativo_X	:= I_XDriveDigitalInput.2;

//Girati
I_ExtraCorsaPositivo_X 	:= I_XDriveDigitalInput.1;
I_ExtraCorsaNegativo_X	:= I_XDriveDigitalInput.2;
I_FermoSicurezzaRilasciato := I_XDriveDigitalInput.3;

I_ExtraCorsaPositivo_Y	:= I_YDriveDigitalInput.1;
I_ExtraCorsaNegativo_Y	:= I_YDriveDigitalInput.2;
I_SicurezzaCinghia_Y 	:=  I_YDriveDigitalInput.3;

I_ExtraCorsaPositivo_Z	:= I_ZDriveDigitalInput.1;
I_ExtraCorsaNegativo_Z	:= I_ZDriveDigitalInput.2;
I_SicurezzaCinghia_Z 	:= I_ZDriveDigitalInput.3;

I_ExtraCorsaPositivo_J 	:=  I_PortQualCiabattaK516_X07.0;
I_ExtraCorsaNegativo_J 	:=  I_PortQualCiabattaK516_X07.1;

I_BascolantePinzaBloccato 	:= I_PortQualCiabattaK516_X08.0;
I_TasteggioCinghiaAsseZ 	:= I_PortQualCiabattaK516_X08.1;

(* Parte a terra *)
//******************** SCHEDA IN AP200.2
I_AutoPal			:= I_AP200_2[1];
I_StartCicloPal	    := I_AP200_2[2];	
I_StopCicloPal	    := I_AP200_2[3];
//I_FREE 		    := I_AP200_2[4];
//I_FREE 			:= I_AP200_2[5];
I_AriaOK		    := I_AP200_2[6];	
I_24VOK_AUXQE	    := I_AP200_2[7];
I_24VOK_SAFETY	    := I_AP200_2[8];
I_24VOK_MONITOR		:= I_AP200_2[9];
I_24VOK_PS305	    := I_AP200_2[10];	
I_24VOK_PS306	    := I_AP200_2[11];
I_24VOK_PS307	    := I_AP200_2[12];
I_24VOK_JB310		:= I_AP200_2[13];
I_24VOK_JB311 	    := I_AP200_2[14];	
I_24VOK_JB312 	    := I_AP200_2[15];
I_24VOK_JB313 	    := I_AP200_2[16];

//******************** SCHEDA IN AP200.5	
I_PresenzaSupporto[1] := I_AP200_5[1];
I_PresenzaTelaio[1]	  := I_AP200_5[2];	
I_PresenzaCentrale[1] := I_AP200_5[3];
I_PresenzaBundle[1]   := I_AP200_5[4];
I_PresenzaSupporto[2] := I_AP200_5[5];
I_PresenzaTelaio[2]	  := I_AP200_5[6];
I_PresenzaCentrale[2] := I_AP200_5[7];
I_PresenzaBundle[2]   := I_AP200_5[8];
I_PresenzaSupporto[3] := I_AP200_5[9];
I_PresenzaTelaio[3]	  := I_AP200_5[10];	
I_PresenzaCentrale[3] := I_AP200_5[11];
I_PresenzaBundle[3]   := I_AP200_5[12];
I_PresenzaSupporto[4] := I_AP200_5[13];
I_PresenzaTelaio[4]	  := I_AP200_5[14];	
I_PresenzaCentrale[4] := I_AP200_5[15];
I_PresenzaBundle[4]   := I_AP200_5[16];

//******************** SCHEDA IN SAFETY AP200.6		
I_RichiestaIngressoConsolle := I_AP200_6[1];
I_ResetRichiestaIngressoConsolle := I_AP200_6[2];
I_PulsanteMarciaConsolle := I_AP200_6[3];
I_RichiestaIngressoPS309 := I_AP200_6[4];

//******************** SCHEDA IN SAFETY AP200.7		
I_RichiestaIngressoPS306 		:= I_AP200_7[1];
I_ResetRichiestaIngressoPS306 	:= I_AP200_7[2];
I_RichiestaIngressoPS307 		:= I_AP200_7[3];
I_ResetRichiestaIngressoPS307 	:= I_AP200_7[4];

//******************** SCHEDA IN AP200.8
//I_FREE 					:= I_AP200_8[1];
//I_FREE 				    := I_AP200_8[2];	
//I_FREE 				    := I_AP200_8[3];
//I_FREE 				    := I_AP200_8[4];
I_24VOK_PS308				:= I_AP200_8[5];
I_24VOK_PS309			    := I_AP200_8[6];	
I_24VOK_JB314			    := I_AP200_8[7];
I_24VOK_JB315			    := I_AP200_8[8];
I_PresenzaSupporto[5]       := I_AP200_8[9];
I_PresenzaTelaio[5]	        := I_AP200_8[10];
I_PresenzaCentrale[5]	    := I_AP200_8[11];
I_PresenzaBundle[5] 	    := I_AP200_8[12];
I_PresenzaSupporto[6]       := I_AP200_8[13];
I_PresenzaTelaio[6]	        := I_AP200_8[14];
I_PresenzaCentrale[6]	    := I_AP200_8[15];
I_PresenzaBundle[6] 	    := I_AP200_8[16];

//******************** SCHEDA IN SAFETY AP200.9	
I_RicevitoreConsensoVeicolo[1] := I_AP200_9[1];
I_RicevitoreConsensoVeicolo[2] := I_AP200_9[2];
I_RicevitoreConsensoVeicolo[3] := I_AP200_9[3];
I_RicevitoreConsensoVeicolo[4] := I_AP200_9[4];

//******************** SCHEDA IN SAFETY AP200.10
I_RichiestaIngressoPS308 		:= I_AP200_10[1];	
I_ResetRichiestaIngressoPS308 	:= I_AP200_10[2];	
//I_BarrieraCentroDx_CH1		:= I_AP200_10[3];	
//I_BarrieraCentroDx_CH2		:= I_AP200_10[4];	

//******************** SCHEDA IN SAFETY AP201.2
//I_FeedBackMarcia				:= I_AP201_12[1];	
I_ResetRichiestaIngressoPS309 	:= I_AP201_2[2];
//I_BarrieraInterna_CH1			:= I_AP201_2[3];
//I_BarrieraInterna_CH2			:= I_AP201_2[4];

//******************** SCHEDA IN AP201.3	
I_PresenzaSupporto[7] 	:= I_AP201_3[1];
I_PresenzaTelaio[7]		:= I_AP201_3[2];	
I_PresenzaCentrale[7]	:= I_AP201_3[3];
I_PresenzaBundle[7] 	:= I_AP201_3[4];
I_PresenzaSupporto[8] 	:= I_AP201_3[5];
I_PresenzaTelaio[8]		:= I_AP201_3[6];	
I_PresenzaCentrale[8]	:= I_AP201_3[7];
I_PresenzaBundle[8] 	:= I_AP201_3[8];
//FREE 					:= I_AP201_3[9];
//FREE 					:= I_AP201_3[10];
//FREE 					:= I_AP201_3[11];
//FREE 					:= I_AP201_3[12];
//FREE 					:= I_AP201_3[13];
//FREE 					:= I_AP201_3[14];
//FREE 					:= I_AP201_3[15];
//FREE 					:= I_AP201_3[16];

//******************** SCHEDA IN SAFETY AP202.2		
I_RicevitoreConsensoVeicolo[5]	:= I_AP202_2[1];	
I_RicevitoreConsensoVeicolo[6] 	:= I_AP202_2[2];	
I_RicevitoreConsensoVeicolo[7]	:= I_AP202_2[3];	
I_RicevitoreConsensoVeicolo[8]	:= I_AP202_2[4];	

//******************** SCHEDA IN SAFETY AP202.3		
I_PresenzaVeicolo[1]	:= I_AP202_3[1];	
I_PresenzaVeicolo[2] 	:= I_AP202_3[2];  
I_PresenzaVeicolo[3]	:= I_AP202_3[3];  
I_PresenzaVeicolo[4]	:= I_AP202_3[4];  

//******************** SCHEDA IN SAFETY AP202.5		
I_PresenzaVeicolo[5]	:= I_AP202_5[1];	
I_PresenzaVeicolo[6] 	:= I_AP202_5[2]; 	
I_PresenzaVeicolo[7]	:= I_AP202_5[3]; 	
I_PresenzaVeicolo[8]	:= I_AP202_5[4]; 	

//******************** SCHEDA IN SAFETY AP202.6		
//I_BarrieraCentroSx_CH1	: BOOL; // 1=
//I_BarrieraCentroSx_CH2 	: BOOL; // 2=	
//I_BarrieraSx_CH1			: BOOL; // 3=	
//I_BarrieraSx_CH2			: BOOL; // 4=	


//FORZATURE


//#######Para Excluir solo simulacion 
IF NOT FROM_HMI_PAL.HMI_AbilitaSimulazioneAVuoto THEN
FOR InPosPx := 1 TO MAXAREAPRESENT DO
	IF I_PresenzaSupporto[InPosPx] OR I_PresenzaBundle[InPosPx]OR I_PresenzaCentrale[InPosPx]  THEN I_PHPresenzaPallet[InPosPx] := TRUE; END_IF
	IF NOT I_PresenzaSupporto[InPosPx] AND NOT I_PresenzaBundle[InPosPx] AND NOT I_PresenzaCentrale[InPosPx] THEN I_PHPresenzaPallet[InPosPx] := FALSE; END_IF	
	
END_FOR
END_IF

(*
I_PHPresenzaPallet[1] := TRUE;
I_PHPresenzaPallet[2] := TRUE;
I_PHPresenzaPallet[3] := FALSE;
I_PHPresenzaPallet[4] := FALSE;
I_PHPresenzaPallet[5] := FALSE;
I_PHPresenzaPallet[6] := FALSE;
I_PHPresenzaPallet[7] := FALSE;
I_PHPresenzaPallet[8] := FALSE;
*)
END_ACTION

ACTION _03_Modules:
(* Test Da ELIMINARE *)
DriveNeedReset := FALSE;
PowerEnableAssi := I_MarciaOK AND NOT DisablePowerPerConfig;
(* Set Stato Emergenze *)
EnablePneumatica := TRUE;

EnableGroupPortSafety := TRUE;

I_BarrierePallettizzatoreOK := (I_SafetyStateBarrierSXPal = 1 AND I_SafetyStateBarrierDXPal = 1 AND I_SafetyStateBarrierCentroDXPal	= 1 AND I_SafetyStateBarrierCentroSXPal	= 1) OR 
								(((I_SafetyStateBarrierDXPal <> 1 OR I_SafetyStateBarrierCentroDXPal <> 1) AND I_SafetyStateBarrierKarv = 1 AND (MachinePalletizerGatesAccess.GateAccessPS308.AccessOK OR MachinePalletizerGatesAccess.GateAccessPS309.AccessOK))OR
								((I_SafetyStateBarrierSXPal <> 1 OR I_SafetyStateBarrierCentroSXPal <> 1) AND I_SafetyStateBarrierKarv = 1 AND (MachinePalletizerGatesAccess.GateAccessPS306.AccessOK OR MachinePalletizerGatesAccess.GateAccessPS307.AccessOK)) OR
								((I_SafetyStateBarrierSXPal <> 1 OR I_SafetyStateBarrierDXPal <> 1 OR I_SafetyStateBarrierCentroSXPal <> 1 OR I_SafetyStateBarrierCentroDXPal <> 1 OR I_SafetyStateBarrierKarv <> 1) AND MachinePalletizerGatesAccess.GateAccessConsolle.AccessOK));							
								
(*I_BarrierePallettizzatoreOK := (I_SafetyStateBarrierSXPal = 1 AND I_SafetyStateBarrierDXPal = 1 AND I_SafetyStateBarrierCentroDXPal	= 1 AND I_SafetyStateBarrierCentroSXPal	= 1) OR 
								((I_SafetyStateBarrierDXPal <> 1 OR I_SafetyStateBarrierCentroDXPal <> 1 AND I_SafetyStateBarrierKarv = 1 AND MachinePalletizerGatesAccess.GateAccessPS308.AccessOK OR MachinePalletizerGatesAccess.GateAccessPS309.AccessOK) OR
								(I_SafetyStateBarrierSXPal <> 1 OR I_SafetyStateBarrierCentroSXPal <> 1 AND I_SafetyStateBarrierKarv = 1 AND MachinePalletizerGatesAccess.GateAccessPS306.AccessOK OR MachinePalletizerGatesAccess.GateAccessPS307.AccessOK) OR
								((I_SafetyStateBarrierSXPal <> 1 OR I_SafetyStateBarrierDXPal <> 1 OR I_SafetyStateBarrierCentroSXPal <> 1 OR I_SafetyStateBarrierCentroDXPal <> 1 OR I_SafetyStateBarrierKarv <> 1) AND MachinePalletizerGatesAccess.GateAccessConsolle.AccessOK));
								*)
							
I_EmergenzeOK := I_SafetyStateEmergenze_Generali = 1 AND 
					I_SafetyStateEmergenza_PS306_307 = 1 AND 
					I_SafetyStateEmergenza_PS308_309 = 1 AND
					I_SafetyStateEmergenze_Generali = 1 AND 
					I_BarrierePallettizzatoreOK;

I_24VAusiliariOK := I_24VOK_AUXQE	AND
                    I_24VOK_SAFETY	AND
                    I_24VOK_MONITOR	AND
                    I_24VOK_PS305	AND
                    I_24VOK_PS306	AND
                    I_24VOK_PS307	AND
                    I_24VOK_JB310	AND
                    I_24VOK_JB311 	AND
                    I_24VOK_JB312 	AND
                    I_24VOK_JB313 	AND
					I_24VOK_PS308   AND
                    I_24VOK_PS309	AND
                    I_24VOK_JB314	AND
                    I_24VOK_JB315;	

IF TEST_ENABLE THEN
	I_ResetAsse_X 		:= FALSE;
	I_ResetAsse_Y 		:= FALSE;
	I_ResetAsse_Z 		:= FALSE;
	DriveNeedReset 		:= FALSE;
	TouchErrorEnable 	:= FALSE;
	SimulaArrayPacchi 	:= TRUE;
END_IF

{region " Macchina "}
(* ******************************************************************************************************** *)
(* INPUT Transfer *)
(* ******************************************************************************************************** *)
(* Machine Palletizer *)
MachinePalletizer_TF.IN.Mode.Auto									:= I_AutoPal;
MachinePalletizer_TF.IN.Mode.Jog 									:= FALSE;
MachinePalletizer_TF.IN.Mode.JogStep 								:= FALSE;
MachinePalletizer_TF.IN.Mode.Man 									:= NOT I_AutoPal;
MachinePalletizer_TF.IN.Mode.Feeding 								:= FALSE;
MachinePalletizer_TF.IN.Mode.Production 							:= FALSE;
MachinePalletizer_TF.IN.Mode.Emptying 								:= FALSE;
MachinePalletizer_TF.IN.Mode.Dry		 							:= FALSE;
MachinePalletizer_TF.IN.Mode.AutoRunRequest							:= I_StartCicloPal AND 
																		NOT MachinePalletizerGatesAccess.GateAccessConsolle.AccesActive AND 
																		NOT MachinePalletizerGatesAccess.GateAccessPS306.AccesActive AND 
																		NOT MachinePalletizerGatesAccess.GateAccessPS307.AccesActive AND 
																		NOT MachinePalletizerGatesAccess.GateAccessPS308.AccesActive AND
																		NOT MachinePalletizerGatesAccess.GateAccessPS309.AccesActive;
																			 
MachinePalletizer_TF.IN.Mode.JogRunRequest							:= FALSE;
MachinePalletizer_TF.IN.Mode.StopRequest							:= NOT I_AutoPal;
MachinePalletizer_TF.IN.Mode.RapidStopRequest						:= I_StopCicloPal;
MachinePalletizer_TF.IN.Mode.ResetRequest							:= I_StartCicloPal;
MachinePalletizer_TF.IN.Mode.PowerOnRequest							:= I_PulsanteMarciaConsolle AND  
																		NOT MachinePalletizerGatesAccess.GateAccessConsolle.AccesActive AND 
																		NOT MachinePalletizerGatesAccess.GateAccessPS306.AccesActive AND 
																		NOT MachinePalletizerGatesAccess.GateAccessPS307.AccesActive AND 
																		NOT MachinePalletizerGatesAccess.GateAccessPS308.AccesActive AND
																		NOT MachinePalletizerGatesAccess.GateAccessPS309.AccesActive;
																			 
MachinePalletizer_TF.IN.Mode.PowerOffRequest						:= FALSE;
MachinePalletizer_TF.IN.Mode.EmergencyRequest						:= NOT I_EmergenzeOK;
MachinePalletizer_TF.IN.PowerOk										:= I_MarciaOK;
MachinePalletizer_TF.IN.SensorAir									:= I_AriaOK;
MachinePalletizer_TF.IN.Sensor24Volt								:= I_24VAusiliariOK;
MachinePalletizer_TF.IN.Y_BeltSafety								:= I_SicurezzaCinghia_Y;
MachinePalletizer_TF.IN.Z_BeltSafety								:= I_SicurezzaCinghia_Z;
MachinePalletizer_TF.IN.PX_GripPresence                             := I_PHPresenzaMaterialePinza;
MachinePalletizer_TF.IN.WD_Trasporti								:= StateETHIPLinea = 0;//Comunicazione con trasporti 

MachinePalletizer_TF.SimulazioneSenzaPalletFalde					:= FROM_HMI_PAL.HMI_AbilitaSimulazioneAVuoto;

MachinePalletizer_TF.AbilitaControlloPHGripPresence					:= FROM_HMI_PAL.HMI_AbilitaControloPXGripPresence AND NOT FROM_HMI_PAL.HMI_AbilitaSimulazioneAVuoto;
//MachinePalletizer_TF.AbilitaControlloCoppia							:= FROM_HMI_PAL.HMI_AbilitaControlloCoppia AND NOT FROM_HMI_PAL.HMI_AbilitaSimulazioneAVuoto;;
MachinePalletizer_TF.AbilitaAnticipoDinamico						:= ADR(FROM_HMI_PAL.HMI_AbilitaAnticipoDinamicoMovimenti);
MachinePalletizer_TF.AbilitaCalcoloIngombroOttimizzato				:= ADR(FROM_HMI_PAL.HMI_AbilitaCalcoloIngombroOttimizzato);
MachinePalletizer_TF.AbilitaDepositoPaccoOrrizzonataleConTasteggio   := ADR(FROM_HMI_PAL.HMI_AbilitaDepositoPaccoOrrizzontaleConTasteggio);
MachinePalletizer_TF.AbilitaInterpolazioneAssi 						:= ADR(FROM_HMI_PAL.HMI_AbilitaInterpolazioneAssi);
MachinePalletizer_TF.STARTInterpolazioneASSI						:= ADR(STARTInterpolazioneASSI);
MachinePalletizer_TF.AbilitaDisposizionePalletContinua 				:= ADR(FROM_HMI_PAL.HMI_AbilitaDepositoPalletContinuo);
MachinePalletizer_TF.AbilitaOffsetInUscitaTasteggioPrelievoPallet   := ADR(FROM_HMI_PAL.HMI_AbilitaOffsetUscitaTasteggioPrelPallet);
MachinePalletizer_TF.AbilitaForzaturaStatoWAMDaCicloRiposoACicloPrelievo  	:=ADR(FROM_HMI_PAL.HMI_AbilitaForzaturaStatoDaRiposoAPrelievo);
MachinePalletizer_TF.AbilitaAccostamentoAsseZ 								:= ADR(FROM_HMI_PAL.HMI_AbilitaAccostamentoAsseZ);
MachinePalletizer_TF.GestioneAZoneAbilitata							:= ADR(FROM_HMI_PAL.HMI_AbilitaGestioneAZone);

MachinePalletizer_TF.Modules										:= ADR(MachinePalletizerModules);	

MachinePalletizer_TF.WorkSpace										:= ADR(WorkSpace);
MachinePalletizer_TF.WorkFootprint									:= ADR(WorkFootprint);
MachinePalletizer_TF.WorkPickPoint									:= ADR(WorkPickPoint);

MachinePalletizer_TF.WorkPickPointState								:= ADR(WorkPickPointState);
MachinePalletizer_TF.WorkPickPointDimension							:= ADR(WorkPickPointDimension);
MachinePalletizer_TF.WorkPickPointOffset							:= ADR(WorkPickPointOffset);
MachinePalletizer_TF.WorkArea										:= ADR(WorkArea);
MachinePalletizer_TF.WorkAreaState									:= ADR(WorkAreaState);
MachinePalletizer_TF.WorkAreaOffset									:= ADR(WorkAreaOffset);
MachinePalletizer_TF.WorkAreaZone								    := ADR(WorkAreaZone);
MachinePalletizer_TF.AxisOverride									:= ADR(AxisOverride);
MachinePalletizer_TF.Pallet											:= ADR(Pallet);
MachinePalletizer_TF.Layer											:= ADR(Layer);
MachinePalletizer_TF.Forming										:= ADR(Forming);
//MachinePalletizer_TF.AxisParK										:= ADR(AxisPar_K);
MachinePalletizer_TF.PickPlaceParameters			 				:= ADR(PickPlaceParameters);
MachinePalletizer_TF.ManCmd											:= ADR(ManCmd);
MachinePalletizer_TF.Mission										:= ADR(Mission);
MachinePalletizer_TF.Traiettoria									:= ADR(Traiettoria);
MachinePalletizer_TF.MachineManCmd 									:= ADR(MachineManCmd);
MachinePalletizer_TF.Cfg.CmdExeCaseEnable 							:= NOT MachinePalletizer_TF.IN.Mode.JogStep;
MachinePalletizer_TF.Cfg.TimeBase 									:= TimeBase;
MachinePalletizer_TF.ProgressiveNrWA								:= ADR(ProgressiveNrWA);
MachinePalletizer_TF.UsedCode										:= ADR(UsedCode);
MachinePalletizer_TF.TCPParameter									:= ADR(TCPParameter);
MachinePalletizer_TF.TilterPack										:= ADR(PaccoSulRibaltino);
MachinePalletizer_TF.PreviousPWA									:= ADR(PreviousPWA);
MachinePalletizer_TF.RestoreCWA										:= ADR(RestoreCWA);
//MachinePalletizer_TF.TouchErrorEnable								:= ADR(TouchErrorEnable);
MachinePalletizer_TF.GateAccesExecuted								:= MachinePalletizerGatesAccess.GateAccessConsolle.AccesActive;// AND MachinePalletizerGatesAccess.GateAccess2.AccesActive;
MachinePalletizer_TF.PreviousStackWA								:= ADR(PreviousStackWA);
MachinePalletizer_TF.WorkAreaManager								:= ADR(WorkAreaManager);
MachinePalletizer_TF.WorkAreaProductionList							:= ADR(WorkAreaProductionList);

MachinePalletizer_TF.RichiestaIngZonaSX := MachinepalletizerGatesAccess.GateAccessPS306.AccessRequest OR MachinepalletizerGatesAccess.GateAccessPS307.AccessRequest;
MachinePalletizer_TF.RichiestaIngZonaDX := MachinepalletizerGatesAccess.GateAccessPS308.AccessRequest OR MachinepalletizerGatesAccess.GateAccessPS309.AccessRequest;		  
			   
//Valuto la posizione in cui sta lavorando il pallettizzatore				
///@@@@@@PortaleADx := MachinePalletizerModules.AX_X.Ax^.Status.ActPosition > 17060;//WorkSpace.X/2;		

///@@@@@@PortaleASx := MachinePalletizerModules.AX_X.Ax^.Status.ActPosition < 17060;//WorkSpace.X/2;					 
							  
IF NOT SimulaArrayPacchi THEN
	MachinePalletizer_TF.ArrayPacchi									:= ADR(I_Trasporti_GEN_OUT_ArrayPacchi);
ELSE
	MachinePalletizer_TF.ArrayPacchi									:= ADR(ArrayPacchiSIMULATO);	
END_IF
MachinePalletizer_TF.MissionStateCase								:= ADR(MissionStateCase);
{endregion}

IF FROM_HMI_PAL.HMI_AbilitaSimulazioneAVuoto THEN
	ProgrammaToModule_X.DisabilitaTasteggio := TRUE;
	ProgrammaToModule_Y.DisabilitaTasteggio := TRUE;
	ProgrammaToModule_Z.DisabilitaTasteggio := TRUE;
	ProgrammaToModule_J.DisabilitaTasteggio := TRUE;
END_IF


(* PX WorkArea *)
IF NOT FROM_HMI_PAL.HMI_AbilitaSimulazioneAVuoto THEN
	FOR i:=1 TO MAXAREAPRESENT DO
		//####################################################
		IF I_PresenzaSupporto[i] OR I_PresenzaBundle[i]OR I_PresenzaCentrale[i]  THEN I_PHPresenzaPallet[i] := TRUE; END_IF
		IF NOT I_PresenzaSupporto[i] AND NOT I_PresenzaBundle[i] AND NOT I_PresenzaCentrale[i] THEN I_PHPresenzaPallet[i] := FALSE; END_IF	
		//####################################################
		MachinePalletizer_TF.IN.PX_WorkArea[i] := I_PHPresenzaPallet[i];
		//MachinePalletizerLGV.PX_WorkArea[i] := I_PHPresenzaPallet[i];
		//MachinePalletizerLGV_NEW.PH_WorkArea[i] := I_PHPresenzaPallet[i];
	END_FOR 
ELSE
	FOR i:=1 TO MAXAREAPRESENT DO
		//######################################################################################
		IF FROM_HMI_PAL.HMI_AbilitaSimulazioneAVuoto AND I_PresenzaSupporto[i] OR I_PresenzaBundle[i] OR I_PresenzaCentrale[i] THEN I_PHPresenzaPalletVirtuale[i] := TRUE; END_IF	
		IF FROM_HMI_PAL.HMI_AbilitaSimulazioneAVuoto AND  NOT I_PresenzaSupporto[i] AND NOT I_PresenzaBundle[i] AND NOT I_PresenzaCentrale[i] THEN I_PHPresenzaPalletVirtuale[i] := FALSE; END_IF	
		//######################################################################################
		MachinePalletizer_TF.IN.PX_WorkArea[i] := I_PHPresenzaPalletVirtuale[i];
		//MachinePalletizerLGV.PX_WorkArea[i] := I_PHPresenzaPallet[i];
		//MachinePalletizerLGV_NEW.PH_WorkArea[i] := I_PHPresenzaPallet[i];
	END_FOR 
END_IF



(*
*)

TFTimerCall(ADR(RetardoFcTastastatore[1]),TimeBase);
TFTimerCall(ADR(RetardoFcTastastatore[2]),TimeBase);
TFTimerCall(ADR(RetardoFcTastastatore[3]),TimeBase);
TFTimerCall(ADR(RetardoFcTastastatore[4]),TimeBase);

TFTimerCall(ADR(RetardoFcTastastatoreJ[1]),TimeBase);
TFTimerCall(ADR(RetardoFcTastastatoreJ[2]),TimeBase);

TFTimerSet(ADR(RetardoFcTastastatore[1]),50, I_TastatorePinza_1);
TFTimerSet(ADR(RetardoFcTastastatore[2]),50, I_TastatorePinza_2);
TFTimerSet(ADR(RetardoFcTastastatore[3]),50,I_TastatorePinza_3);
TFTimerSet(ADR(RetardoFcTastastatore[4]),50, I_TastatorePinza_4);

TFTimerSet(ADR(RetardoFcTastastatoreJ[1]),200,I_TastatorePinza_1);
TFTimerSet(ADR(RetardoFcTastastatoreJ[2]),200,I_TastatorePinza_2);

TFTimerCall(ADR(Re_TastatoreEmergenzaPinza[1]),TimeBase);
TFTimerCall(ADR(Re_TastatoreEmergenzaPinza[2]),TimeBase);
TFTimerCall(ADR(Re_TastatoreEmergenzaPinza[3]),TimeBase);
TFTimerCall(ADR(Re_TastatoreEmergenzaPinza[4]),TimeBase);

TFTimerSet(ADR(Re_TastatoreEmergenzaPinza[1]),50,I_TastatoreEmergenzaPinza_1);
TFTimerSet(ADR(Re_TastatoreEmergenzaPinza[2]),50,I_TastatoreEmergenzaPinza_2);
TFTimerSet(ADR(Re_TastatoreEmergenzaPinza[3]),50,I_TastatoreEmergenzaPinza_3);
TFTimerSet(ADR(Re_TastatoreEmergenzaPinza[4]),50 ,I_TastatoreEmergenzaPinza_4);



RetardoTastatore :=  NOT TFTimerDone(ADR(RetardoFcTastastatore[1]))
						AND NOT TFTimerDone(ADR(RetardoFcTastastatore[2]))
							AND NOT TFTimerDone(ADR(RetardoFcTastastatore[3]))
								AND NOT TFTimerDone(ADR(RetardoFcTastastatore[4]));                   //   OR TFTimerDone(ADR(RetardoFcTastastatore[2])) OR TFTimerDone(ADR(RetardoFcTastastatore[3]) OR TFTimerDone(ADR(RetardoFcTastastatore[4])) ;
Temp_Bool[5] := NOT TFTimerDone(ADR(RetardoFcTastastatore[1]))
						AND NOT TFTimerDone(ADR(RetardoFcTastastatore[4]));
Temp_Bool[6] := NOT  TFTimerDone(ADR(RetardoFcTastastatore[2]))
						AND NOT TFTimerDone(ADR(RetardoFcTastastatore[3]));
						
Re_In_TastatorePinza[1] 	 := NOT TFTimerDone(ADR(RetardoFcTastastatore[1]));	
Re_In_TastatorePinza[2] 	 := NOT TFTimerDone(ADR(RetardoFcTastastatore[2]));	
Re_In_TastatorePinza[3] 	 := NOT TFTimerDone(ADR(RetardoFcTastastatore[3]));	
Re_In_TastatorePinza[4] 	 := NOT TFTimerDone(ADR(RetardoFcTastastatore[4]));						
						
Re_In_TastatoreEmergenzaPinza[1] :=  NOT TFTimerDone(ADR(Re_TastatoreEmergenzaPinza[1])) ;
Re_In_TastatoreEmergenzaPinza[2] :=  NOT TFTimerDone(ADR(Re_TastatoreEmergenzaPinza[2])) ;
Re_In_TastatoreEmergenzaPinza[3] :=  NOT TFTimerDone(ADR(Re_TastatoreEmergenzaPinza[3])) ;
Re_In_TastatoreEmergenzaPinza[4] :=  NOT TFTimerDone(ADR(Re_TastatoreEmergenzaPinza[4])) ;


Fun_SensoresTasteggio(
	Sensor_Tasteo_1:= I_TastatorePinza_1 , 
	Sensor_Tasteo_2:= I_TastatorePinza_2 , 
	Sensor_Tasteo_3:= I_TastatorePinza_3 , 
	Sensor_Tasteo_4:= I_TastatorePinza_4 , 
	Nu_sensores_Dar_Out:= 4 , 
	Sensores_Tasteggio_Ok=> Ok_sensores_Tastator , 
	Nu_Sesores_Activos=> Nu_Sensores_Leyendo);


(* Valorizzo la presenza delle falde *)

(************************************************************************
******************************* MODULO X ********************************
************************************************************************)
(* Configurazione Asse X *)

MachinePalletizerModules.AX_X.Ax 							:= ADR(X_AxisLib);
MachinePalletizerModules.AX_X.Ax^.AxRef 					:= ADR(X_Axis);
MachinePalletizerModules.AX_X.Ax^.TimeBase 					:= TimeBase;
MachinePalletizerModules.AX_X.Ax^.PowerEnable 				:= PowerEnableAssi;
MachinePalletizerModules.AX_X.Ax^.PowerEnablePositive   	:= PowerEnableAssi AND (I_ExtraCorsaPositivo_X OR NOT TouchErrorEnable);
MachinePalletizerModules.AX_X.Ax^.PowerEnableNegative   	:= PowerEnableAssi AND (I_ExtraCorsaNegativo_X OR NOT TouchErrorEnable);
MachinePalletizerModules.AX_X.Ax^.EncoderType				:= ABSOLUTE_ENCODER;
MachinePalletizerModules.AX_X.AxHomingParameters			:= ADR(AxisHomingParameters_X);


